LIN {X 0,Y 516.467,Z 235.214,A -85,B 0,C 180,E1 -4935.822,E2 -4935.822} C_VEL
LIN {X 0,Y 516.489,Z 231.626,A -85,B 0,C 180,E1 -4939.019,E2 -4939.019} C_VEL
LIN {X 0,Y 516.548,Z 228.079,A -85,B 0,C 180,E1 -4942.181,E2 -4942.181} C_VEL
LIN {X 0,Y 516.558,Z 225.48,A -85,B 0,C 180,E1 -4944.536,E2 -4944.536} C_VEL
LIN {X 0,Y 516.606,Z 224.598,A -85,B 0,C 180,E1 -4945.319,E2 -4945.319} C_VEL
LIN {X 0,Y 516.602,Z 224.14,A -85,B 0,C 180,E1 -4946.1,E2 -4946.1} C_VEL
LIN {X 0,Y 516.939,Z 224.095,A -85,B 0,C 180,E1 -4948.443,E2 -4948.443} C_VEL
LIN {X 0,Y 517.084,Z 224.078,A -85,B 0,C 180,E1 -4950.78,E2 -4950.78} C_VEL
LIN {X 0,Y 517.003,Z 224.088,A -85,B 0,C 180,E1 -4953.118,E2 -4953.118} C_VEL
LIN {X 0,Y 516.997,Z 224.088,A -85,B 0,C 180,E1 -4956.244,E2 -4956.244} C_VEL
LIN {X 0,Y 516.948,Z 224.094,A -85,B 0,C 180,E1 -4959.39,E2 -4959.39} C_VEL
LIN {X 0,Y 516.969,Z 224.092,A -85,B 0,C 180,E1 -4961.825,E2 -4961.825} C_VEL
LIN {X 0,Y 516.931,Z 224.096,A -85,B 0,C 180,E1 -4965.148,E2 -4965.148} C_VEL
LIN {X 0,Y 516.914,Z 224.097,A -85,B 0,C 180,E1 -4968.223,E2 -4968.223} C_VEL
LIN {X 0,Y 516.903,Z 224.099,A -85,B 0,C 180,E1 -4970.703,E2 -4970.703} C_VEL
LIN {X 0,Y 516.881,Z 224.103,A -85,B 0,C 180,E1 -4973.224,E2 -4973.224} C_VEL
LIN {X 0,Y 516.934,Z 224.095,A -85,B 0,C 180,E1 -4976.198,E2 -4976.198} C_VEL
LIN {X 0,Y 516.912,Z 224.098,A -85,B 0,C 180,E1 -4979.306,E2 -4979.306} C_VEL
LIN {X 0,Y 516.892,Z 224.101,A -85,B 0,C 180,E1 -4982.546,E2 -4982.546} C_VEL
LIN {X 0,Y 516.875,Z 224.102,A -85,B 0,C 180,E1 -4985.334,E2 -4985.334} C_VEL
LIN {X 0,Y 516.874,Z 224.101,A -85,B 0,C 180,E1 -4987.945,E2 -4987.945} C_VEL
LIN {X 0,Y 516.897,Z 224.101,A -85,B 0,C 180,E1 -4990.741,E2 -4990.741} C_VEL
LIN {X 0,Y 516.877,Z 224.102,A -85,B 0,C 180,E1 -4993.905,E2 -4993.905} C_VEL
LIN {X 0,Y 516.877,Z 224.102,A -85,B 0,C 180,E1 -4996.109,E2 -4996.109} C_VEL
LIN {X 0,Y 516.9,Z 224.098,A -85,B 0,C 180,E1 -4999.262,E2 -4999.262} C_VEL
LIN {X 0,Y 516.878,Z 224.103,A -85,B 0,C 180,E1 -5002.058,E2 -5002.058} C_VEL
LIN {X 0,Y 516.89,Z 224.1,A -85,B 0,C 180,E1 -5005.178,E2 -5005.178} C_VEL
LIN {X 0,Y 516.875,Z 224.104,A -85,B 0,C 180,E1 -5007.977,E2 -5007.977} C_VEL
LIN {X 0,Y 516.921,Z 224.096,A -85,B 0,C 180,E1 -5010.697,E2 -5010.697} C_VEL
LIN {X 0,Y 516.943,Z 224.095,A -85,B 0,C 180,E1 -5013.806,E2 -5013.806} C_VEL
LIN {X 0,Y 516.861,Z 224.106,A -85,B 0,C 180,E1 -5016.778,E2 -5016.778} C_VEL
LIN {X 0,Y 516.942,Z 224.094,A -85,B 0,C 180,E1 -5019.733,E2 -5019.733} C_VEL
LIN {X 0,Y 516.922,Z 224.098,A -85,B 0,C 180,E1 -5022.597,E2 -5022.597} C_VEL
LIN {X 0,Y 516.946,Z 224.094,A -85,B 0,C 180,E1 -5025.032,E2 -5025.032} C_VEL
LIN {X 0,Y 517.01,Z 224.087,A -85,B 0,C 180,E1 -5028.236,E2 -5028.236} C_VEL
LIN {X 0,Y 516.96,Z 224.091,A -85,B 0,C 180,E1 -5031.401,E2 -5031.401} C_VEL
LIN {X 0,Y 517.015,Z 224.085,A -85,B 0,C 180,E1 -5033.758,E2 -5033.758} C_VEL
LIN {X 0,Y 517.085,Z 224.078,A -85,B 0,C 180,E1 -5037.664,E2 -5037.664} C_VEL
LIN {X 0,Y 517.098,Z 224.075,A -85,B 0,C 180,E1 -5040.78,E2 -5040.78} C_VEL
LIN {X 0,Y 516.992,Z 224.087,A -85,B 0,C 180,E1 -5043.118,E2 -5043.118} C_VEL
LIN {X 0,Y 517.008,Z 224.086,A -85,B 0,C 180,E1 -5046.244,E2 -5046.244} C_VEL
LIN {X 0,Y 516.949,Z 224.094,A -85,B 0,C 180,E1 -5049.39,E2 -5049.39} C_VEL
LIN {X 0,Y 516.961,Z 224.092,A -85,B 0,C 180,E1 -5051.808,E2 -5051.808} C_VEL
LIN {X 0,Y 516.952,Z 224.093,A -85,B 0,C 180,E1 -5055.146,E2 -5055.146} C_VEL
LIN {X 0,Y 516.921,Z 224.097,A -85,B 0,C 180,E1 -5058.223,E2 -5058.223} C_VEL
LIN {X 0,Y 516.921,Z 224.098,A -85,B 0,C 180,E1 -5060.702,E2 -5060.702} C_VEL
LIN {X 0,Y 516.894,Z 224.1,A -85,B 0,C 180,E1 -5064.074,E2 -5064.074} C_VEL
LIN {X 0,Y 516.915,Z 224.097,A -85,B 0,C 180,E1 -5066.659,E2 -5066.659} C_VEL
LIN {X 0,Y 516.918,Z 224.099,A -85,B 0,C 180,E1 -5069.524,E2 -5069.524} C_VEL
LIN {X 0,Y 516.903,Z 224.098,A -85,B 0,C 180,E1 -5072.543,E2 -5072.543} C_VEL
LIN {X 0,Y 516.874,Z 224.105,A -85,B 0,C 180,E1 -5075.33,E2 -5075.33} C_VEL
LIN {X 0,Y 516.888,Z 224.1,A -85,B 0,C 180,E1 -5077.943,E2 -5077.943} C_VEL
LIN {X 0,Y 516.892,Z 224.1,A -85,B 0,C 180,E1 -5080.742,E2 -5080.742} C_VEL
LIN {X 0,Y 516.891,Z 224.1,A -85,B 0,C 180,E1 -5082.832,E2 -5082.832} C_VEL
LIN {X 0,Y 516.904,Z 224.097,A -85,B 0,C 180,E1 -5085.007,E2 -5085.007} C_VEL
LIN {X 0,Y 516.922,Z 224.096,A -85,B 0,C 180,E1 -5088.399,E2 -5088.399} C_VEL
LIN {X 0,Y 516.91,Z 224.226,A -85,B 0,C 180,E1 -5091.385,E2 -5091.385} C_VEL
LIN {X 0,Y 517.907,Z 230.288,A -85,B 0,C 180,E1 -5093.821,E2 -5093.821} C_VEL
LIN {X 0,Y 517.949,Z 235.762,A -85,B 0,C 180,E1 -5095.865,E2 -5095.865} C_VEL
LIN {X 0,Y 517.702,Z 243.001,A -85,B 0,C 180,E1 -5098.462,E2 -5098.462} C_VEL
LIN {X 0,Y 517.337,Z 252.149,A -85,B 0,C 180,E1 -5101.609,E2 -5101.609} C_VEL
LIN {X 0,Y 517.129,Z 261.34,A -85,B 0,C 180,E1 -5104.652,E2 -5104.652} C_VEL
LIN {X 0,Y 516.921,Z 270.537,A -85,B 0,C 180,E1 -5107.623,E2 -5107.623} C_VEL
LIN {X 0,Y 516.769,Z 279.876,A -85,B 0,C 180,E1 -5110.536,E2 -5110.536} C_VEL
LIN {X 0,Y 516.6,Z 290.693,A -85,B 0,C 180,E1 -5113.805,E2 -5113.805} C_VEL
LIN {X 0,Y 516.522,Z 298.272,A -85,B 0,C 180,E1 -5116.099,E2 -5116.099} C_VEL
LIN {X 0,Y 518.346,Z 310.965,A -85,B 0,C 180,E1 -5116.436,E2 -5116.436} C_VEL
LIN {X 0,Y 518.162,Z 323.395,A -85,B 0,C 180,E1 -5116.868,E2 -5116.868} C_VEL
LIN {X 0,Y 517.868,Z 335.653,A -85,B 0,C 180,E1 -5117.458,E2 -5117.458} C_VEL
LIN {X 0,Y 517.559,Z 346.352,A -85,B 0,C 180,E1 -5118.121,E2 -5118.121} C_VEL
LIN {X 0,Y 517.314,Z 356.898,A -85,B 0,C 180,E1 -5118.936,E2 -5118.936} C_VEL
LIN {X 0,Y 517.031,Z 366.256,A -85,B 0,C 180,E1 -5119.821,E2 -5119.821} C_VEL
LIN {X 0,Y 516.801,Z 374.794,A -85,B 0,C 180,E1 -5120.805,E2 -5120.805} C_VEL
LIN {X 0,Y 516.587,Z 383.122,A -85,B 0,C 180,E1 -5121.983,E2 -5121.983} C_VEL
LIN {X 0,Y 516.441,Z 390.084,A -85,B 0,C 180,E1 -5123.208,E2 -5123.208} C_VEL
LIN {X 0,Y 516.397,Z 395.989,A -85,B 0,C 180,E1 -5124.532,E2 -5124.532} C_VEL
LIN {X 0,Y 516.314,Z 399.982,A -85,B 0,C 180,E1 -5125.706,E2 -5125.706} C_VEL
LIN {X 0,Y 516.283,Z 402.931,A -85,B 0,C 180,E1 -5126.878,E2 -5126.878} C_VEL
LIN {X 0,Y 516.262,Z 404.335,A -85,B 0,C 180,E1 -5127.659,E2 -5127.659} C_VEL
LIN {X 0,Y 516.166,Z 405.942,A -85,B 0,C 180,E1 -5129.219,E2 -5129.219} C_VEL
LIN {X 0,Y 516.166,Z 406.157,A -85,B 0,C 180,E1 -5129.999,E2 -5129.999} C_VEL
LIN {X 0,Y 516.192,Z 405.326,A -85,B 0,C 180,E1 -5131.56,E2 -5131.56} C_VEL
LIN {X 0,Y 516.262,Z 404.325,A -85,B 0,C 180,E1 -5132.34,E2 -5132.34} C_VEL
LIN {X 0,Y 516.283,Z 402.917,A -85,B 0,C 180,E1 -5133.121,E2 -5133.121} C_VEL
LIN {X 0,Y 516.313,Z 399.957,A -85,B 0,C 180,E1 -5134.293,E2 -5134.293} C_VEL
LIN {X 0,Y 516.397,Z 395.952,A -85,B 0,C 180,E1 -5135.466,E2 -5135.466} C_VEL
LIN {X 0,Y 516.473,Z 390.048,A -85,B 0,C 180,E1 -5136.788,E2 -5136.788} C_VEL
LIN {X 0,Y 516.586,Z 383.063,A -85,B 0,C 180,E1 -5138.015,E2 -5138.015} C_VEL
LIN {X 0,Y 516.8,Z 374.717,A -85,B 0,C 180,E1 -5139.194,E2 -5139.194} C_VEL
LIN {X 0,Y 517,Z 366.163,A -85,B 0,C 180,E1 -5140.178,E2 -5140.178} C_VEL
LIN {X 0,Y 517.346,Z 355.609,A -85,B 0,C 180,E1 -5141.161,E2 -5141.161} C_VEL
LIN {X 0,Y 517.589,Z 343.972,A -85,B 0,C 180,E1 -5142.033,E2 -5142.033} C_VEL
LIN {X 0,Y 517.92,Z 331.793,A -85,B 0,C 180,E1 -5142.738,E2 -5142.738} C_VEL
LIN {X 0,Y 518.206,Z 319.398,A -85,B 0,C 180,E1 -5143.279,E2 -5143.279} C_VEL
LIN {X 0,Y 518.231,Z 310.339,A -85,B 0,C 180,E1 -5143.578,E2 -5143.578} C_VEL
LIN {X 0,Y 516.503,Z 297.887,A -85,B 0,C 180,E1 -5143.925,E2 -5143.925} C_VEL
LIN {X 0,Y 516.582,Z 288.976,A -85,B 0,C 180,E1 -5146.6,E2 -5146.6} C_VEL
LIN {X 0,Y 516.745,Z 279.489,A -85,B 0,C 180,E1 -5149.463,E2 -5149.463} C_VEL
LIN {X 0,Y 516.901,Z 269.991,A -85,B 0,C 180,E1 -5152.397,E2 -5152.397} C_VEL
LIN {X 0,Y 517.058,Z 260.81,A -85,B 0,C 180,E1 -5155.35,E2 -5155.35} C_VEL
LIN {X 0,Y 517.258,Z 251.656,A -85,B 0,C 180,E1 -5158.394,E2 -5158.394} C_VEL
LIN {X 0,Y 517.556,Z 243.591,A -85,B 0,C 180,E1 -5161.185,E2 -5161.185} C_VEL
LIN {X 0,Y 517.842,Z 236.392,A -85,B 0,C 180,E1 -5163.809,E2 -5163.809} C_VEL
LIN {X 0,Y 518.004,Z 231.462,A -85,B 0,C 180,E1 -5165.689,E2 -5165.689} C_VEL
LIN {X 0,Y 517.334,Z 226.619,A -85,B 0,C 180,E1 -5167.684,E2 -5167.684} C_VEL
LIN {X 0,Y 516.882,Z 224.103,A -85,B 0,C 180,E1 -5168.834,E2 -5168.834} C_VEL
LIN {X 0,Y 516.915,Z 224.098,A -85,B 0,C 180,E1 -5171.774,E2 -5171.774} C_VEL
LIN {X 0,Y 516.894,Z 224.101,A -85,B 0,C 180,E1 -5175.006,E2 -5175.006} C_VEL
LIN {X 0,Y 516.916,Z 224.098,A -85,B 0,C 180,E1 -5178.397,E2 -5178.397} C_VEL
LIN {X 0,Y 516.88,Z 224.103,A -85,B 0,C 180,E1 -5181.283,E2 -5181.283} C_VEL
LIN {X 0,Y 516.886,Z 224.102,A -85,B 0,C 180,E1 -5184.22,E2 -5184.22} C_VEL
LIN {X 0,Y 516.894,Z 224.101,A -85,B 0,C 180,E1 -5187.052,E2 -5187.052} C_VEL
LIN {X 0,Y 516.889,Z 224.101,A -85,B 0,C 180,E1 -5189.795,E2 -5189.795} C_VEL
LIN {X 0,Y 516.927,Z 224.098,A -85,B 0,C 180,E1 -5192.466,E2 -5192.466} C_VEL
LIN {X 0,Y 516.872,Z 224.103,A -85,B 0,C 180,E1 -5195.069,E2 -5195.069} C_VEL
LIN {X 0,Y 516.865,Z 224.103,A -85,B 0,C 180,E1 -5197.62,E2 -5197.62} C_VEL
LIN {X 0,Y 516.929,Z 224.096,A -85,B 0,C 180,E1 -5200.129,E2 -5200.129} C_VEL
LIN {X 0,Y 516.926,Z 224.098,A -85,B 0,C 180,E1 -5202.595,E2 -5202.595} C_VEL
LIN {X 0,Y 516.938,Z 224.096,A -85,B 0,C 180,E1 -5205.029,E2 -5205.029} C_VEL
LIN {X 0,Y 517,Z 224.089,A -85,B 0,C 180,E1 -5208.233,E2 -5208.233} C_VEL
LIN {X 0,Y 516.965,Z 224.092,A -85,B 0,C 180,E1 -5211.399,E2 -5211.399} C_VEL
LIN {X 0,Y 517.007,Z 224.087,A -85,B 0,C 180,E1 -5213.756,E2 -5213.756} C_VEL
LIN {X 0,Y 517.077,Z 224.078,A -85,B 0,C 180,E1 -5217.662,E2 -5217.662} C_VEL
LIN {X 0,Y 517.09,Z 224.078,A -85,B 0,C 180,E1 -5220.778,E2 -5220.778} C_VEL
LIN {X 0,Y 517.01,Z 224.087,A -85,B 0,C 180,E1 -5223.116,E2 -5223.116} C_VEL
LIN {X 0,Y 517.004,Z 224.088,A -85,B 0,C 180,E1 -5226.242,E2 -5226.242} C_VEL
LIN {X 0,Y 516.953,Z 224.093,A -85,B 0,C 180,E1 -5229.388,E2 -5229.388} C_VEL
LIN {X 0,Y 516.975,Z 224.091,A -85,B 0,C 180,E1 -5231.823,E2 -5231.823} C_VEL
LIN {X 0,Y 516.935,Z 224.097,A -85,B 0,C 180,E1 -5235.145,E2 -5235.145} C_VEL
LIN {X 0,Y 516.859,Z 224.108,A -85,B 0,C 180,E1 -5237.86,E2 -5237.86} C_VEL
LIN {X 0,Y 516.643,Z 224.391,A -85,B 0,C 180,E1 -5239.88,E2 -5239.88} C_VEL
LIN {X 0,Y 516.601,Z 227.102,A -85,B 0,C 180,E1 -5242.389,E2 -5242.389} C_VEL
LIN {X 0,Y 516.556,Z 229.906,A -85,B 0,C 180,E1 -5244.945,E2 -5244.945} C_VEL
LIN {X 0,Y 516.491,Z 233.036,A -85,B 0,C 180,E1 -5247.816,E2 -5247.816} C_VEL
LIN {X 0,Y 516.431,Z 236.511,A -85,B 0,C 180,E1 -5250.981,E2 -5250.981} C_VEL
LIN {X 0,Y 516.357,Z 239.775,A -85,B 0,C 180,E1 -5253.918,E2 -5253.918} C_VEL
LIN {X 0,Y 516.278,Z 242.962,A -85,B 0,C 180,E1 -5256.794,E2 -5256.794} C_VEL
LIN {X 0,Y 516.297,Z 245.663,A -85,B 0,C 180,E1 -5259.199,E2 -5259.199} C_VEL
LIN {X 0,Y 518.486,Z 256.449,A -85,B 0,C 180,E1 -5259.549,E2 -5259.549} C_VEL
LIN {X 0,Y 518.293,Z 269.265,A -85,B 0,C 180,E1 -5260.032,E2 -5260.032} C_VEL
LIN {X 0,Y 517.996,Z 281.061,A -85,B 0,C 180,E1 -5260.633,E2 -5260.633} C_VEL
LIN {X 0,Y 517.716,Z 291.239,A -85,B 0,C 180,E1 -5261.298,E2 -5261.298} C_VEL
LIN {X 0,Y 517.48,Z 301.242,A -85,B 0,C 180,E1 -5262.109,E2 -5262.109} C_VEL
LIN {X 0,Y 517.178,Z 310.969,A -85,B 0,C 180,E1 -5263.08,E2 -5263.08} C_VEL
LIN {X 0,Y 516.902,Z 319.892,A -85,B 0,C 180,E1 -5264.177,E2 -5264.177} C_VEL
LIN {X 0,Y 516.877,Z 320.67,A -85,B 0,C 180,E1 -5264.286,E2 -5264.286} C_VEL
LIN {X 0,Y 516.11,Z 324.315,A -85,B 0,C 180,E1 -5264.8,E2 -5264.8} C_VEL
LIN {X 0,Y 511.766,Z 331.837,A -85,B 0,C 180,E1 -5266.008,E2 -5266.008} C_VEL
LIN {X 0,Y 509.733,Z 335.586,A -85,B 0,C 180,E1 -5266.757,E2 -5266.757} C_VEL
LIN {X 0,Y 509.375,Z 337.272,A -85,B 0,C 180,E1 -5267.155,E2 -5267.155} C_VEL
LIN {X 0,Y 509.29,Z 342.03,A -85,B 0,C 180,E1 -5268.519,E2 -5268.519} C_VEL
LIN {X 0,Y 509.243,Z 344.721,A -85,B 0,C 180,E1 -5269.562,E2 -5269.562} C_VEL
LIN {X 0,Y 509.148,Z 346.72,A -85,B 0,C 180,E1 -5270.621,E2 -5270.621} C_VEL
LIN {X 0,Y 509.089,Z 348.144,A -85,B 0,C 180,E1 -5271.893,E2 -5271.893} C_VEL
LIN {X 0,Y 509.085,Z 348.541,A -85,B 0,C 180,E1 -5273.194,E2 -5273.194} C_VEL
LIN {X 0,Y 509.077,Z 347.811,A -85,B 0,C 180,E1 -5274.563,E2 -5274.563} C_VEL
LIN {X 0,Y 509.164,Z 345.936,A -85,B 0,C 180,E1 -5275.909,E2 -5275.909} C_VEL
LIN {X 0,Y 509.23,Z 342.382,A -85,B 0,C 180,E1 -5277.437,E2 -5277.437} C_VEL
LIN {X 0,Y 509.359,Z 337.714,A -85,B 0,C 180,E1 -5278.807,E2 -5278.807} C_VEL
LIN {X 0,Y 509.544,Z 331.262,A -85,B 0,C 180,E1 -5280.23,E2 -5280.23} C_VEL
LIN {X 0,Y 509.748,Z 324.793,A -85,B 0,C 180,E1 -5281.355,E2 -5281.355} C_VEL
LIN {X 0,Y 509.989,Z 316.614,A -85,B 0,C 180,E1 -5282.507,E2 -5282.507} C_VEL
LIN {X 0,Y 510.276,Z 307.618,A -85,B 0,C 180,E1 -5283.535,E2 -5283.535} C_VEL
LIN {X 0,Y 510.638,Z 296.904,A -85,B 0,C 180,E1 -5284.527,E2 -5284.527} C_VEL
LIN {X 0,Y 510.951,Z 285.423,A -85,B 0,C 180,E1 -5285.367,E2 -5285.367} C_VEL
LIN {X 0,Y 511.25,Z 272.908,A -85,B 0,C 180,E1 -5286.077,E2 -5286.077} C_VEL
LIN {X 0,Y 511.593,Z 260.24,A -85,B 0,C 180,E1 -5286.604,E2 -5286.604} C_VEL
LIN {X 0,Y 511.386,Z 255.913,A -85,B 0,C 180,E1 -5286.755,E2 -5286.755} C_VEL
LIN {X 0,Y 509.252,Z 245.771,A -85,B 0,C 180,E1 -5287.081,E2 -5287.081} C_VEL
LIN {X 0,Y 509.288,Z 242.619,A -85,B 0,C 180,E1 -5289.82,E2 -5289.82} C_VEL
LIN {X 0,Y 509.338,Z 239.772,A -85,B 0,C 180,E1 -5292.329,E2 -5292.329} C_VEL
LIN {X 0,Y 509.409,Z 236.06,A -85,B 0,C 180,E1 -5295.622,E2 -5295.622} C_VEL
LIN {X 0,Y 509.422,Z 232.451,A -85,B 0,C 180,E1 -5298.864,E2 -5298.864} C_VEL
LIN {X 0,Y 509.487,Z 228.868,A -85,B 0,C 180,E1 -5302.072,E2 -5302.072} C_VEL
LIN {X 0,Y 509.488,Z 226.23,A -85,B 0,C 180,E1 -5304.46,E2 -5304.46} C_VEL
LIN {X 0,Y 509.545,Z 225.354,A -85,B 0,C 180,E1 -5305.254,E2 -5305.254} C_VEL
LIN {X 0,Y 509.597,Z 225.012,A -85,B 0,C 180,E1 -5306.838,E2 -5306.838} C_VEL
LIN {X 0,Y 509.904,Z 224.971,A -85,B 0,C 180,E1 -5308.421,E2 -5308.421} C_VEL
LIN {X 0,Y 510.053,Z 224.954,A -85,B 0,C 180,E1 -5310.79,E2 -5310.79} C_VEL
LIN {X 0,Y 509.945,Z 224.967,A -85,B 0,C 180,E1 -5313.161,E2 -5313.161} C_VEL
LIN {X 0,Y 509.965,Z 224.963,A -85,B 0,C 180,E1 -5316.331,E2 -5316.331} C_VEL
LIN {X 0,Y 509.907,Z 224.972,A -85,B 0,C 180,E1 -5318.721,E2 -5318.721} C_VEL
LIN {X 0,Y 509.937,Z 224.967,A -85,B 0,C 180,E1 -5321.932,E2 -5321.932} C_VEL
LIN {X 0,Y 509.88,Z 224.975,A -85,B 0,C 180,E1 -5325.243,E2 -5325.243} C_VEL
LIN {X 0,Y 509.876,Z 224.974,A -85,B 0,C 180,E1 -5328.002,E2 -5328.002} C_VEL
LIN {X 0,Y 509.846,Z 224.979,A -85,B 0,C 180,E1 -5331.003,E2 -5331.003} C_VEL
LIN {X 0,Y 509.839,Z 224.979,A -85,B 0,C 180,E1 -5333.564,E2 -5333.564} C_VEL
LIN {X 0,Y 509.903,Z 224.97,A -85,B 0,C 180,E1 -5336.381,E2 -5336.381} C_VEL
LIN {X 0,Y 509.867,Z 224.976,A -85,B 0,C 180,E1 -5338.846,E2 -5338.846} C_VEL
LIN {X 0,Y 509.816,Z 224.982,A -85,B 0,C 180,E1 -5341.591,E2 -5341.591} C_VEL
LIN {X 0,Y 509.846,Z 224.978,A -85,B 0,C 180,E1 -5344.415,E2 -5344.415} C_VEL
LIN {X 0,Y 509.811,Z 224.982,A -85,B 0,C 180,E1 -5347.342,E2 -5347.342} C_VEL
LIN {X 0,Y 509.854,Z 224.977,A -85,B 0,C 180,E1 -5350.382,E2 -5350.382} C_VEL
LIN {X 0,Y 509.834,Z 224.98,A -85,B 0,C 180,E1 -5353.066,E2 -5353.066} C_VEL
LIN {X 0,Y 509.825,Z 224.98,A -85,B 0,C 180,E1 -5355.794,E2 -5355.794} C_VEL
LIN {X 0,Y 509.861,Z 224.978,A -85,B 0,C 180,E1 -5358.577,E2 -5358.577} C_VEL
LIN {X 0,Y 509.855,Z 224.975,A -85,B 0,C 180,E1 -5361.665,E2 -5361.665} C_VEL
LIN {X 0,Y 509.841,Z 224.979,A -85,B 0,C 180,E1 -5364.625,E2 -5364.625} C_VEL
LIN {X 0,Y 509.861,Z 224.975,A -85,B 0,C 180,E1 -5367.483,E2 -5367.483} C_VEL
LIN {X 0,Y 509.857,Z 224.978,A -85,B 0,C 180,E1 -5370.275,E2 -5370.275} C_VEL
LIN {X 0,Y 509.885,Z 224.972,A -85,B 0,C 180,E1 -5372.946,E2 -5372.946} C_VEL
LIN {X 0,Y 509.852,Z 224.976,A -85,B 0,C 180,E1 -5375.575,E2 -5375.575} C_VEL
LIN {X 0,Y 509.824,Z 224.983,A -85,B 0,C 180,E1 -5378.15,E2 -5378.15} C_VEL
LIN {X 0,Y 509.866,Z 224.975,A -85,B 0,C 180,E1 -5380.683,E2 -5380.683} C_VEL
LIN {X 0,Y 509.882,Z 224.972,A -85,B 0,C 180,E1 -5383.176,E2 -5383.176} C_VEL
LIN {X 0,Y 509.868,Z 224.975,A -85,B 0,C 180,E1 -5385.636,E2 -5385.636} C_VEL
LIN {X 0,Y 509.926,Z 224.966,A -85,B 0,C 180,E1 -5388.876,E2 -5388.876} C_VEL
LIN {X 0,Y 509.926,Z 224.969,A -85,B 0,C 180,E1 -5392.079,E2 -5392.079} C_VEL
LIN {X 0,Y 509.986,Z 224.96,A -85,B 0,C 180,E1 -5394.466,E2 -5394.466} C_VEL
LIN {X 0,Y 510.057,Z 224.954,A -85,B 0,C 180,E1 -5397.632,E2 -5397.632} C_VEL
LIN {X 0,Y 510.062,Z 224.952,A -85,B 0,C 180,E1 -5400.001,E2 -5400.001} C_VEL
LIN {X 0,Y 510.057,Z 224.951,A -85,B 0,C 180,E1 -5402.37,E2 -5402.37} C_VEL
LIN {X 0,Y 509.959,Z 224.964,A -85,B 0,C 180,E1 -5406.331,E2 -5406.331} C_VEL
LIN {X 0,Y 509.912,Z 224.969,A -85,B 0,C 180,E1 -5408.721,E2 -5408.721} C_VEL
LIN {X 0,Y 509.913,Z 224.97,A -85,B 0,C 180,E1 -5411.933,E2 -5411.933} C_VEL
LIN {X 0,Y 509.903,Z 224.971,A -85,B 0,C 180,E1 -5415.243,E2 -5415.243} C_VEL
LIN {X 0,Y 509.866,Z 224.975,A -85,B 0,C 180,E1 -5418.485,E2 -5418.485} C_VEL
LIN {X 0,Y 509.859,Z 224.976,A -85,B 0,C 180,E1 -5421.002,E2 -5421.002} C_VEL
LIN {X 0,Y 509.828,Z 224.981,A -85,B 0,C 180,E1 -5423.565,E2 -5423.565} C_VEL
LIN {X 0,Y 509.883,Z 224.974,A -85,B 0,C 180,E1 -5427.057,E2 -5427.057} C_VEL
LIN {X 0,Y 509.866,Z 224.975,A -85,B 0,C 180,E1 -5429.751,E2 -5429.751} C_VEL
LIN {X 0,Y 509.876,Z 224.974,A -85,B 0,C 180,E1 -5432.773,E2 -5432.773} C_VEL
LIN {X 0,Y 509.834,Z 224.979,A -85,B 0,C 180,E1 -5435.578,E2 -5435.578} C_VEL
LIN {X 0,Y 509.857,Z 224.975,A -85,B 0,C 180,E1 -5438.338,E2 -5438.338} C_VEL
LIN {X 0,Y 509.864,Z 224.975,A -85,B 0,C 180,E1 -5441.426,E2 -5441.426} C_VEL
LIN {X 0,Y 509.848,Z 224.978,A -85,B 0,C 180,E1 -5444.67,E2 -5444.67} C_VEL
LIN {X 0,Y 509.864,Z 224.975,A -85,B 0,C 180,E1 -5448.103,E2 -5448.103} C_VEL
LIN {X 0,Y 509.879,Z 225.144,A -85,B 0,C 180,E1 -5451.158,E2 -5451.158} C_VEL
LIN {X 0,Y 510.933,Z 231.463,A -85,B 0,C 180,E1 -5453.737,E2 -5453.737} C_VEL
LIN {X 0,Y 510.988,Z 236.566,A -85,B 0,C 180,E1 -5455.673,E2 -5455.673} C_VEL
LIN {X 0,Y 510.686,Z 244.227,A -85,B 0,C 180,E1 -5458.469,E2 -5458.469} C_VEL
LIN {X 0,Y 510.378,Z 251.989,A -85,B 0,C 180,E1 -5461.186,E2 -5461.186} C_VEL
LIN {X 0,Y 510.125,Z 261.115,A -85,B 0,C 180,E1 -5464.279,E2 -5464.279} C_VEL
LIN {X 0,Y 509.881,Z 270.771,A -85,B 0,C 180,E1 -5467.445,E2 -5467.445} C_VEL
LIN {X 0,Y 509.715,Z 279.602,A -85,B 0,C 180,E1 -5470.256,E2 -5470.256} C_VEL
LIN {X 0,Y 509.533,Z 290.304,A -85,B 0,C 180,E1 -5473.574,E2 -5473.574} C_VEL
LIN {X 0,Y 509.424,Z 297.841,A -85,B 0,C 180,E1 -5475.901,E2 -5475.901} C_VEL
LIN {X 0,Y 511.3,Z 310.989,A -85,B 0,C 180,E1 -5476.258,E2 -5476.258} C_VEL
LIN {X 0,Y 511.352,Z 319.154,A -85,B 0,C 180,E1 -5476.538,E2 -5476.538} C_VEL
LIN {X 0,Y 510.987,Z 331.525,A -85,B 0,C 180,E1 -5477.085,E2 -5477.085} C_VEL
LIN {X 0,Y 510.695,Z 342.32,A -85,B 0,C 180,E1 -5477.71,E2 -5477.71} C_VEL
LIN {X 0,Y 510.412,Z 352.944,A -85,B 0,C 180,E1 -5478.482,E2 -5478.482} C_VEL
LIN {X 0,Y 510.069,Z 363.893,A -85,B 0,C 180,E1 -5479.48,E2 -5479.48} C_VEL
LIN {X 0,Y 509.789,Z 372.791,A -85,B 0,C 180,E1 -5480.477,E2 -5480.477} C_VEL
LIN {X 0,Y 509.575,Z 381.48,A -85,B 0,C 180,E1 -5481.673,E2 -5481.673} C_VEL
LIN {X 0,Y 509.41,Z 388.422,A -85,B 0,C 180,E1 -5482.867,E2 -5482.867} C_VEL
LIN {X 0,Y 509.314,Z 393.988,A -85,B 0,C 180,E1 -5484.059,E2 -5484.059} C_VEL
LIN {X 0,Y 509.187,Z 398.35,A -85,B 0,C 180,E1 -5485.249,E2 -5485.249} C_VEL
LIN {X 0,Y 509.276,Z 400.666,A -85,B 0,C 180,E1 -5486.043,E2 -5486.043} C_VEL
LIN {X 0,Y 509.202,Z 402.535,A -85,B 0,C 180,E1 -5486.834,E2 -5486.834} C_VEL
LIN {X 0,Y 509.191,Z 403.94,A -85,B 0,C 180,E1 -5487.626,E2 -5487.626} C_VEL
LIN {X 0,Y 509.079,Z 405.544,A -85,B 0,C 180,E1 -5489.208,E2 -5489.208} C_VEL
LIN {X 0,Y 509.078,Z 405.759,A -85,B 0,C 180,E1 -5489.999,E2 -5489.999} C_VEL
LIN {X 0,Y 509.113,Z 404.926,A -85,B 0,C 180,E1 -5491.581,E2 -5491.581} C_VEL
LIN {X 0,Y 509.19,Z 403.923,A -85,B 0,C 180,E1 -5492.372,E2 -5492.372} C_VEL
LIN {X 0,Y 509.202,Z 402.511,A -85,B 0,C 180,E1 -5493.164,E2 -5493.164} C_VEL
LIN {X 0,Y 509.207,Z 399.546,A -85,B 0,C 180,E1 -5494.353,E2 -5494.353} C_VEL
LIN {X 0,Y 509.309,Z 395.538,A -85,B 0,C 180,E1 -5495.542,E2 -5495.542} C_VEL
LIN {X 0,Y 509.408,Z 389.475,A -85,B 0,C 180,E1 -5496.913,E2 -5496.913} C_VEL
LIN {X 0,Y 509.509,Z 382.635,A -85,B 0,C 180,E1 -5498.127,E2 -5498.127} C_VEL
LIN {X 0,Y 509.744,Z 374.284,A -85,B 0,C 180,E1 -5499.322,E2 -5499.322} C_VEL
LIN {X 0,Y 509.972,Z 365.724,A -85,B 0,C 180,E1 -5500.32,E2 -5500.32} C_VEL
LIN {X 0,Y 510.356,Z 355.163,A -85,B 0,C 180,E1 -5501.316,E2 -5501.316} C_VEL
LIN {X 0,Y 510.599,Z 343.519,A -85,B 0,C 180,E1 -5502.2,E2 -5502.2} C_VEL
LIN {X 0,Y 510.988,Z 331.333,A -85,B 0,C 180,E1 -5502.914,E2 -5502.914} C_VEL
LIN {X 0,Y 511.305,Z 318.936,A -85,B 0,C 180,E1 -5503.462,E2 -5503.462} C_VEL
LIN {X 0,Y 511.27,Z 310.779,A -85,B 0,C 180,E1 -5503.741,E2 -5503.741} C_VEL
LIN {X 0,Y 509.507,Z 298.545,A -85,B 0,C 180,E1 -5504.079,E2 -5504.079} C_VEL
LIN {X 0,Y 509.42,Z 297.45,A -85,B 0,C 180,E1 -5504.123,E2 -5504.123} C_VEL
LIN {X 0,Y 509.513,Z 288.533,A -85,B 0,C 180,E1 -5506.837,E2 -5506.837} C_VEL
LIN {X 0,Y 509.671,Z 279.113,A -85,B 0,C 180,E1 -5509.744,E2 -5509.744} C_VEL
LIN {X 0,Y 509.852,Z 269.739,A -85,B 0,C 180,E1 -5512.703,E2 -5512.703} C_VEL
LIN {X 0,Y 510.03,Z 260.498,A -85,B 0,C 180,E1 -5515.724,E2 -5515.724} C_VEL
LIN {X 0,Y 510.288,Z 251.466,A -85,B 0,C 180,E1 -5518.818,E2 -5518.818} C_VEL
LIN {X 0,Y 510.609,Z 243.801,A -85,B 0,C 180,E1 -5521.535,E2 -5521.535} C_VEL
LIN {X 0,Y 510.923,Z 236.159,A -85,B 0,C 180,E1 -5524.377,E2 -5524.377} C_VEL
LIN {X 0,Y 510.932,Z 231.414,A -85,B 0,C 180,E1 -5526.261,E2 -5526.261} C_VEL
LIN {X 0,Y 509.865,Z 224.978,A -85,B 0,C 180,E1 -5529.063,E2 -5529.063} C_VEL
LIN {X 0,Y 509.859,Z 224.978,A -85,B 0,C 180,E1 -5531.896,E2 -5531.896} C_VEL
LIN {X 0,Y 509.838,Z 224.98,A -85,B 0,C 180,E1 -5535.329,E2 -5535.329} C_VEL
LIN {X 0,Y 509.858,Z 224.978,A -85,B 0,C 180,E1 -5538.574,E2 -5538.574} C_VEL
LIN {X 0,Y 509.85,Z 224.978,A -85,B 0,C 180,E1 -5541.785,E2 -5541.785} C_VEL
LIN {X 0,Y 509.842,Z 224.98,A -85,B 0,C 180,E1 -5544.622,E2 -5544.622} C_VEL
LIN {X 0,Y 509.861,Z 224.976,A -85,B 0,C 180,E1 -5547.48,E2 -5547.48} C_VEL
LIN {X 0,Y 509.856,Z 224.978,A -85,B 0,C 180,E1 -5550.273,E2 -5550.273} C_VEL
LIN {X 0,Y 509.883,Z 224.973,A -85,B 0,C 180,E1 -5552.943,E2 -5552.943} C_VEL
LIN {X 0,Y 509.848,Z 224.979,A -85,B 0,C 180,E1 -5555.572,E2 -5555.572} C_VEL
LIN {X 0,Y 509.819,Z 224.983,A -85,B 0,C 180,E1 -5558.147,E2 -5558.147} C_VEL
LIN {X 0,Y 509.861,Z 224.976,A -85,B 0,C 180,E1 -5560.68,E2 -5560.68} C_VEL
LIN {X 0,Y 509.881,Z 224.973,A -85,B 0,C 180,E1 -5563.174,E2 -5563.174} C_VEL
LIN {X 0,Y 509.861,Z 224.976,A -85,B 0,C 180,E1 -5565.633,E2 -5565.633} C_VEL
LIN {X 0,Y 509.918,Z 224.968,A -85,B 0,C 180,E1 -5568.874,E2 -5568.874} C_VEL
LIN {X 0,Y 509.947,Z 224.965,A -85,B 0,C 180,E1 -5572.077,E2 -5572.077} C_VEL
LIN {X 0,Y 509.979,Z 224.961,A -85,B 0,C 180,E1 -5574.463,E2 -5574.463} C_VEL
LIN {X 0,Y 510.049,Z 224.953,A -85,B 0,C 180,E1 -5577.63,E2 -5577.63} C_VEL
LIN {X 0,Y 510.06,Z 224.953,A -85,B 0,C 180,E1 -5580.788,E2 -5580.788} C_VEL
LIN {X 0,Y 509.952,Z 224.966,A -85,B 0,C 180,E1 -5583.159,E2 -5583.159} C_VEL
LIN {X 0,Y 509.972,Z 224.965,A -85,B 0,C 180,E1 -5586.328,E2 -5586.328} C_VEL
LIN {X 0,Y 509.912,Z 224.971,A -85,B 0,C 180,E1 -5588.719,E2 -5588.719} C_VEL
LIN {X 0,Y 509.943,Z 224.967,A -85,B 0,C 180,E1 -5591.929,E2 -5591.929} C_VEL
LIN {X 0,Y 509.884,Z 224.976,A -85,B 0,C 180,E1 -5595.241,E2 -5595.241} C_VEL
LIN {X 0,Y 509.79,Z 224.988,A -85,B 0,C 180,E1 -5597.969,E2 -5597.969} C_VEL
LIN {X 0,Y 509.618,Z 225.01,A -85,B 0,C 180,E1 -5599.327,E2 -5599.327} C_VEL
LIN {X 0,Y 509.567,Z 225.636,A -85,B 0,C 180,E1 -5600.307,E2 -5600.307} C_VEL
LIN {X 0,Y 509.52,Z 229.172,A -85,B 0,C 180,E1 -5603.577,E2 -5603.577} C_VEL
LIN {X 0,Y 509.441,Z 232.062,A -85,B 0,C 180,E1 -5606.273,E2 -5606.273} C_VEL
LIN {X 0,Y 509.392,Z 234.863,A -85,B 0,C 180,E1 -5608.872,E2 -5608.872} C_VEL
LIN {X 0,Y 509.336,Z 237.916,A -85,B 0,C 180,E1 -5611.622,E2 -5611.622} C_VEL
LIN {X 0,Y 509.261,Z 241.014,A -85,B 0,C 180,E1 -5614.457,E2 -5614.457} C_VEL
LIN {X 0,Y 509.198,Z 244.313,A -85,B 0,C 180,E1 -5617.392,E2 -5617.392} C_VEL
LIN {X 0,Y 509.204,Z 246.111,A -85,B 0,C 180,E1 -5619.011,E2 -5619.011} C_VEL
LIN {X 0,Y 511.562,Z 257.166,A -85,B 0,C 180,E1 -5619.375,E2 -5619.375} C_VEL
LIN {X 0,Y 511.38,Z 270.454,A -85,B 0,C 180,E1 -5619.89,E2 -5619.89} C_VEL
LIN {X 0,Y 511.072,Z 282.72,A -85,B 0,C 180,E1 -5620.54,E2 -5620.54} C_VEL
LIN {X 0,Y 510.699,Z 294.274,A -85,B 0,C 180,E1 -5621.34,E2 -5621.34} C_VEL
LIN {X 0,Y 510.391,Z 305.142,A -85,B 0,C 180,E1 -5622.287,E2 -5622.287} C_VEL
LIN {X 0,Y 510.077,Z 314.944,A -85,B 0,C 180,E1 -5623.36,E2 -5623.36} C_VEL
LIN {X 0,Y 509.804,Z 323.211,A -85,B 0,C 180,E1 -5624.477,E2 -5624.477} C_VEL
LIN {X 0,Y 509.555,Z 331.168,A -85,B 0,C 180,E1 -5625.822,E2 -5625.822} C_VEL
LIN {X 0,Y 509.375,Z 337.272,A -85,B 0,C 180,E1 -5627.155,E2 -5627.155} C_VEL
LIN {X 0,Y 508.655,Z 339.636,A -85,B 0,C 180,E1 -5627.761,E2 -5627.761} C_VEL
LIN {X 0,Y 505.722,Z 343.049,A -85,B 0,C 180,E1 -5628.76,E2 -5628.76} C_VEL
LIN {X 0,Y 503.251,Z 345.255,A -85,B 0,C 180,E1 -5629.583,E2 -5629.583} C_VEL
LIN {X 0,Y 502.166,Z 346.546,A -85,B 0,C 180,E1 -5630.231,E2 -5630.231} C_VEL
LIN {X 0,Y 502.065,Z 346.895,A -85,B 0,C 180,E1 -5630.453,E2 -5630.453} C_VEL
LIN {X 0,Y 502,Z 348.602,A -85,B 0,C 180,E1 -5631.976,E2 -5631.976} C_VEL
LIN {X 0,Y 501.992,Z 348.958,A -85,B 0,C 180,E1 -5632.987,E2 -5632.987} C_VEL
LIN {X 0,Y 501.988,Z 348.478,A -85,B 0,C 180,E1 -5634.29,E2 -5634.29} C_VEL
LIN {X 0,Y 502.072,Z 346.82,A -85,B 0,C 180,E1 -5635.675,E2 -5635.675} C_VEL
LIN {X 0,Y 502.154,Z 343.798,A -85,B 0,C 180,E1 -5637.109,E2 -5637.109} C_VEL
LIN {X 0,Y 502.274,Z 339.206,A -85,B 0,C 180,E1 -5638.595,E2 -5638.595} C_VEL
LIN {X 0,Y 502.414,Z 334.396,A -85,B 0,C 180,E1 -5639.764,E2 -5639.764} C_VEL
LIN {X 0,Y 502.594,Z 328.426,A -85,B 0,C 180,E1 -5640.928,E2 -5640.928} C_VEL
LIN {X 0,Y 502.876,Z 321.098,A -85,B 0,C 180,E1 -5642.085,E2 -5642.085} C_VEL
LIN {X 0,Y 503.154,Z 312.195,A -85,B 0,C 180,E1 -5643.22,E2 -5643.22} C_VEL
LIN {X 0,Y 503.536,Z 302.193,A -85,B 0,C 180,E1 -5644.253,E2 -5644.253} C_VEL
LIN {X 0,Y 503.842,Z 291.403,A -85,B 0,C 180,E1 -5645.148,E2 -5645.148} C_VEL
LIN {X 0,Y 504.229,Z 279.184,A -85,B 0,C 180,E1 -5645.941,E2 -5645.941} C_VEL
LIN {X 0,Y 504.544,Z 266.733,A -85,B 0,C 180,E1 -5646.557,E2 -5646.557} C_VEL
LIN {X 0,Y 504.563,Z 257.315,A -85,B 0,C 180,E1 -5646.908,E2 -5646.908} C_VEL
LIN {X 0,Y 502.173,Z 246.113,A -85,B 0,C 180,E1 -5647.297,E2 -5647.297} C_VEL
LIN {X 0,Y 502.213,Z 242.6,A -85,B 0,C 180,E1 -5650.376,E2 -5650.376} C_VEL
LIN {X 0,Y 502.252,Z 239.729,A -85,B 0,C 180,E1 -5652.912,E2 -5652.912} C_VEL
LIN {X 0,Y 502.318,Z 236.921,A -85,B 0,C 180,E1 -5655.414,E2 -5655.414} C_VEL
LIN {X 0,Y 502.362,Z 233.257,A -85,B 0,C 180,E1 -5658.706,E2 -5658.706} C_VEL
LIN {X 0,Y 502.418,Z 229.663,A -85,B 0,C 180,E1 -5661.96,E2 -5661.96} C_VEL
LIN {X 0,Y 502.503,Z 227.87,A -85,B 0,C 180,E1 -5663.577,E2 -5663.577} C_VEL
LIN {X 0,Y 502.486,Z 226.126,A -85,B 0,C 180,E1 -5665.187,E2 -5665.187} C_VEL
LIN {X 0,Y 502.869,Z 225.847,A -85,B 0,C 180,E1 -5668.399,E2 -5668.399} C_VEL
LIN {X 0,Y 503.023,Z 225.829,A -85,B 0,C 180,E1 -5670.801,E2 -5670.801} C_VEL
LIN {X 0,Y 502.889,Z 225.845,A -85,B 0,C 180,E1 -5673.205,E2 -5673.205} C_VEL
LIN {X 0,Y 502.915,Z 225.842,A -85,B 0,C 180,E1 -5676.42,E2 -5676.42} C_VEL
LIN {X 0,Y 502.865,Z 225.849,A -85,B 0,C 180,E1 -5678.844,E2 -5678.844} C_VEL
LIN {X 0,Y 502.88,Z 225.846,A -85,B 0,C 180,E1 -5682.102,E2 -5682.102} C_VEL
LIN {X 0,Y 502.835,Z 225.853,A -85,B 0,C 180,E1 -5685.401,E2 -5685.401} C_VEL
LIN {X 0,Y 502.834,Z 225.851,A -85,B 0,C 180,E1 -5688.124,E2 -5688.124} C_VEL
LIN {X 0,Y 502.785,Z 225.858,A -85,B 0,C 180,E1 -5691.312,E2 -5691.312} C_VEL
LIN {X 0,Y 502.791,Z 225.855,A -85,B 0,C 180,E1 -5693.915,E2 -5693.915} C_VEL
LIN {X 0,Y 502.87,Z 225.847,A -85,B 0,C 180,E1 -5696.567,E2 -5696.567} C_VEL
LIN {X 0,Y 502.814,Z 225.854,A -85,B 0,C 180,E1 -5699.289,E2 -5699.289} C_VEL
LIN {X 0,Y 502.779,Z 225.857,A -85,B 0,C 180,E1 -5702.086,E2 -5702.086} C_VEL
LIN {X 0,Y 502.802,Z 225.857,A -85,B 0,C 180,E1 -5704.966,E2 -5704.966} C_VEL
LIN {X 0,Y 502.787,Z 225.856,A -85,B 0,C 180,E1 -5707.955,E2 -5707.955} C_VEL
LIN {X 0,Y 502.82,Z 225.853,A -85,B 0,C 180,E1 -5711.067,E2 -5711.067} C_VEL
LIN {X 0,Y 502.776,Z 225.857,A -85,B 0,C 180,E1 -5713.377,E2 -5713.377} C_VEL
LIN {X 0,Y 502.784,Z 225.857,A -85,B 0,C 180,E1 -5715.663,E2 -5715.663} C_VEL
LIN {X 0,Y 502.822,Z 225.852,A -85,B 0,C 180,E1 -5719.006,E2 -5719.006} C_VEL
LIN {X 0,Y 502.794,Z 225.857,A -85,B 0,C 180,E1 -5722.048,E2 -5722.048} C_VEL
LIN {X 0,Y 502.806,Z 225.854,A -85,B 0,C 180,E1 -5725.037,E2 -5725.037} C_VEL
LIN {X 0,Y 502.783,Z 225.859,A -85,B 0,C 180,E1 -5727.917,E2 -5727.917} C_VEL
LIN {X 0,Y 502.823,Z 225.853,A -85,B 0,C 180,E1 -5730.714,E2 -5730.714} C_VEL
LIN {X 0,Y 502.863,Z 225.848,A -85,B 0,C 180,E1 -5733.441,E2 -5733.441} C_VEL
LIN {X 0,Y 502.776,Z 225.86,A -85,B 0,C 180,E1 -5736.087,E2 -5736.087} C_VEL
LIN {X 0,Y 502.785,Z 225.857,A -85,B 0,C 180,E1 -5738.691,E2 -5738.691} C_VEL
LIN {X 0,Y 502.832,Z 225.851,A -85,B 0,C 180,E1 -5741.25,E2 -5741.25} C_VEL
LIN {X 0,Y 502.822,Z 225.854,A -85,B 0,C 180,E1 -5743.769,E2 -5743.769} C_VEL
LIN {X 0,Y 502.835,Z 225.852,A -85,B 0,C 180,E1 -5746.256,E2 -5746.256} C_VEL
LIN {X 0,Y 502.897,Z 225.842,A -85,B 0,C 180,E1 -5748.719,E2 -5748.719} C_VEL
LIN {X 0,Y 502.885,Z 225.847,A -85,B 0,C 180,E1 -5751.968,E2 -5751.968} C_VEL
LIN {X 0,Y 502.942,Z 225.837,A -85,B 0,C 180,E1 -5754.388,E2 -5754.388} C_VEL
LIN {X 0,Y 503.027,Z 225.829,A -85,B 0,C 180,E1 -5757.599,E2 -5757.599} C_VEL
LIN {X 0,Y 503.033,Z 225.828,A -85,B 0,C 180,E1 -5760.001,E2 -5760.001} C_VEL
LIN {X 0,Y 503.026,Z 225.826,A -85,B 0,C 180,E1 -5762.403,E2 -5762.403} C_VEL
LIN {X 0,Y 502.938,Z 225.841,A -85,B 0,C 180,E1 -5765.615,E2 -5765.615} C_VEL
LIN {X 0,Y 502.888,Z 225.845,A -85,B 0,C 180,E1 -5768.035,E2 -5768.035} C_VEL
LIN {X 0,Y 502.885,Z 225.846,A -85,B 0,C 180,E1 -5771.284,E2 -5771.284} C_VEL
LIN {X 0,Y 502.849,Z 225.849,A -85,B 0,C 180,E1 -5774.572,E2 -5774.572} C_VEL
LIN {X 0,Y 502.826,Z 225.853,A -85,B 0,C 180,E1 -5777.909,E2 -5777.909} C_VEL
LIN {X 0,Y 502.839,Z 225.851,A -85,B 0,C 180,E1 -5780.537,E2 -5780.537} C_VEL
LIN {X 0,Y 502.796,Z 225.857,A -85,B 0,C 180,E1 -5783.041,E2 -5783.041} C_VEL
LIN {X 0,Y 502.854,Z 225.849,A -85,B 0,C 180,E1 -5786.557,E2 -5786.557} C_VEL
LIN {X 0,Y 502.832,Z 225.852,A -85,B 0,C 180,E1 -5789.288,E2 -5789.288} C_VEL
LIN {X 0,Y 502.791,Z 225.856,A -85,B 0,C 180,E1 -5792.085,E2 -5792.085} C_VEL
LIN {X 0,Y 502.804,Z 225.855,A -85,B 0,C 180,E1 -5794.966,E2 -5794.966} C_VEL
LIN {X 0,Y 502.801,Z 225.854,A -85,B 0,C 180,E1 -5797.954,E2 -5797.954} C_VEL
LIN {X 0,Y 502.829,Z 225.855,A -85,B 0,C 180,E1 -5801.066,E2 -5801.066} C_VEL
LIN {X 0,Y 502.795,Z 225.857,A -85,B 0,C 180,E1 -5804.53,E2 -5804.53} C_VEL
LIN {X 0,Y 502.804,Z 225.855,A -85,B 0,C 180,E1 -5807.86,E2 -5807.86} C_VEL
LIN {X 0,Y 502.847,Z 226.003,A -85,B 0,C 180,E1 -5810.898,E2 -5810.898} C_VEL
LIN {X 0,Y 503.941,Z 232.503,A -85,B 0,C 180,E1 -5813.604,E2 -5813.604} C_VEL
LIN {X 0,Y 504.024,Z 237.01,A -85,B 0,C 180,E1 -5815.355,E2 -5815.355} C_VEL
LIN {X 0,Y 503.701,Z 245.05,A -85,B 0,C 180,E1 -5818.334,E2 -5818.334} C_VEL
LIN {X 0,Y 503.304,Z 254.262,A -85,B 0,C 180,E1 -5821.609,E2 -5821.609} C_VEL
LIN {X 0,Y 503.039,Z 263.513,A -85,B 0,C 180,E1 -5824.778,E2 -5824.778} C_VEL
LIN {X 0,Y 502.776,Z 272.717,A -85,B 0,C 180,E1 -5827.825,E2 -5827.825} C_VEL
LIN {X 0,Y 502.607,Z 281.929,A -85,B 0,C 180,E1 -5830.815,E2 -5830.815} C_VEL
LIN {X 0,Y 502.443,Z 292.571,A -85,B 0,C 180,E1 -5834.171,E2 -5834.171} C_VEL
LIN {X 0,Y 502.354,Z 297.456,A -85,B 0,C 180,E1 -5835.698,E2 -5835.698} C_VEL
LIN {X 0,Y 504.258,Z 311.009,A -85,B 0,C 180,E1 -5836.075,E2 -5836.075} C_VEL
LIN {X 0,Y 504.483,Z 315.262,A -85,B 0,C 180,E1 -5836.223,E2 -5836.223} C_VEL
LIN {X 0,Y 504.151,Z 328.129,A -85,B 0,C 180,E1 -5836.753,E2 -5836.753} C_VEL
LIN {X 0,Y 503.77,Z 340.585,A -85,B 0,C 180,E1 -5837.453,E2 -5837.453} C_VEL
LIN {X 0,Y 503.412,Z 351.256,A -85,B 0,C 180,E1 -5838.218,E2 -5838.218} C_VEL
LIN {X 0,Y 503.12,Z 361.519,A -85,B 0,C 180,E1 -5839.129,E2 -5839.129} C_VEL
LIN {X 0,Y 502.806,Z 370.749,A -85,B 0,C 180,E1 -5840.14,E2 -5840.14} C_VEL
LIN {X 0,Y 502.515,Z 379.742,A -85,B 0,C 180,E1 -5841.352,E2 -5841.352} C_VEL
LIN {X 0,Y 502.351,Z 386.988,A -85,B 0,C 180,E1 -5842.564,E2 -5842.564} C_VEL
LIN {X 0,Y 502.238,Z 391.879,A -85,B 0,C 180,E1 -5843.572,E2 -5843.572} C_VEL
LIN {X 0,Y 502.18,Z 396.634,A -85,B 0,C 180,E1 -5844.78,E2 -5844.78} C_VEL
LIN {X 0,Y 502.167,Z 400.269,A -85,B 0,C 180,E1 -5845.987,E2 -5845.987} C_VEL
LIN {X 0,Y 502.124,Z 402.14,A -85,B 0,C 180,E1 -5846.79,E2 -5846.79} C_VEL
LIN {X 0,Y 502.122,Z 403.546,A -85,B 0,C 180,E1 -5847.593,E2 -5847.593} C_VEL
LIN {X 0,Y 501.996,Z 405.148,A -85,B 0,C 180,E1 -5849.197,E2 -5849.197} C_VEL
LIN {X 0,Y 501.992,Z 405.361,A -85,B 0,C 180,E1 -5849.999,E2 -5849.999} C_VEL
LIN {X 0,Y 502.037,Z 404.526,A -85,B 0,C 180,E1 -5851.604,E2 -5851.604} C_VEL
LIN {X 0,Y 502.121,Z 403.521,A -85,B 0,C 180,E1 -5852.406,E2 -5852.406} C_VEL
LIN {X 0,Y 502.123,Z 402.106,A -85,B 0,C 180,E1 -5853.209,E2 -5853.209} C_VEL
LIN {X 0,Y 502.106,Z 399.135,A -85,B 0,C 180,E1 -5854.414,E2 -5854.414} C_VEL
LIN {X 0,Y 502.221,Z 395.124,A -85,B 0,C 180,E1 -5855.621,E2 -5855.621} C_VEL
LIN {X 0,Y 502.334,Z 389.054,A -85,B 0,C 180,E1 -5857.011,E2 -5857.011} C_VEL
LIN {X 0,Y 502.46,Z 382.209,A -85,B 0,C 180,E1 -5858.242,E2 -5858.242} C_VEL
LIN {X 0,Y 502.692,Z 373.85,A -85,B 0,C 180,E1 -5859.454,E2 -5859.454} C_VEL
LIN {X 0,Y 502.96,Z 365.285,A -85,B 0,C 180,E1 -5860.465,E2 -5860.465} C_VEL
LIN {X 0,Y 503.365,Z 354.717,A -85,B 0,C 180,E1 -5861.475,E2 -5861.475} C_VEL
LIN {X 0,Y 503.629,Z 343.29,A -85,B 0,C 180,E1 -5862.355,E2 -5862.355} C_VEL
LIN {X 0,Y 503.981,Z 332.822,A -85,B 0,C 180,E1 -5862.994,E2 -5862.994} C_VEL
LIN {X 0,Y 504.319,Z 321.069,A -85,B 0,C 180,E1 -5863.549,E2 -5863.549} C_VEL
LIN {X 0,Y 504.333,Z 311.57,A -85,B 0,C 180,E1 -5863.895,E2 -5863.895} C_VEL
LIN {X 0,Y 502.509,Z 298.623,A -85,B 0,C 180,E1 -5864.27,E2 -5864.27} C_VEL
LIN {X 0,Y 502.349,Z 297.013,A -85,B 0,C 180,E1 -5864.326,E2 -5864.326} C_VEL
LIN {X 0,Y 502.437,Z 288.127,A -85,B 0,C 180,E1 -5867.081,E2 -5867.081} C_VEL
LIN {X 0,Y 502.648,Z 278.783,A -85,B 0,C 180,E1 -5870.032,E2 -5870.032} C_VEL
LIN {X 0,Y 502.8,Z 269.498,A -85,B 0,C 180,E1 -5873.039,E2 -5873.039} C_VEL
LIN {X 0,Y 503.034,Z 260.29,A -85,B 0,C 180,E1 -5876.109,E2 -5876.109} C_VEL
LIN {X 0,Y 503.299,Z 251.28,A -85,B 0,C 180,E1 -5879.257,E2 -5879.257} C_VEL
LIN {X 0,Y 503.652,Z 243.666,A -85,B 0,C 180,E1 -5882.022,E2 -5882.022} C_VEL
LIN {X 0,Y 504.02,Z 236.226,A -85,B 0,C 180,E1 -5884.868,E2 -5884.868} C_VEL
LIN {X 0,Y 504.021,Z 233.336,A -85,B 0,C 180,E1 -5886.026,E2 -5886.026} C_VEL
LIN {X 0,Y 503.119,Z 227.592,A -85,B 0,C 180,E1 -5888.531,E2 -5888.531} C_VEL
LIN {X 0,Y 502.824,Z 225.854,A -85,B 0,C 180,E1 -5889.36,E2 -5889.36} C_VEL
LIN {X 0,Y 502.802,Z 225.858,A -85,B 0,C 180,E1 -5892.198,E2 -5892.198} C_VEL
LIN {X 0,Y 502.784,Z 225.859,A -85,B 0,C 180,E1 -5895.469,E2 -5895.469} C_VEL
LIN {X 0,Y 502.82,Z 225.855,A -85,B 0,C 180,E1 -5898.933,E2 -5898.933} C_VEL
LIN {X 0,Y 502.792,Z 225.859,A -85,B 0,C 180,E1 -5902.045,E2 -5902.045} C_VEL
LIN {X 0,Y 502.807,Z 225.855,A -85,B 0,C 180,E1 -5905.034,E2 -5905.034} C_VEL
LIN {X 0,Y 502.782,Z 225.86,A -85,B 0,C 180,E1 -5907.914,E2 -5907.914} C_VEL
LIN {X 0,Y 502.822,Z 225.853,A -85,B 0,C 180,E1 -5910.711,E2 -5910.711} C_VEL
LIN {X 0,Y 502.86,Z 225.85,A -85,B 0,C 180,E1 -5913.438,E2 -5913.438} C_VEL
LIN {X 0,Y 502.772,Z 225.86,A -85,B 0,C 180,E1 -5916.084,E2 -5916.084} C_VEL
LIN {X 0,Y 502.78,Z 225.857,A -85,B 0,C 180,E1 -5918.688,E2 -5918.688} C_VEL
LIN {X 0,Y 502.827,Z 225.853,A -85,B 0,C 180,E1 -5921.247,E2 -5921.247} C_VEL
LIN {X 0,Y 502.819,Z 225.855,A -85,B 0,C 180,E1 -5923.766,E2 -5923.766} C_VEL
LIN {X 0,Y 502.828,Z 225.853,A -85,B 0,C 180,E1 -5926.254,E2 -5926.254} C_VEL
LIN {X 0,Y 502.888,Z 225.844,A -85,B 0,C 180,E1 -5928.716,E2 -5928.716} C_VEL
LIN {X 0,Y 502.897,Z 225.844,A -85,B 0,C 180,E1 -5931.965,E2 -5931.965} C_VEL
LIN {X 0,Y 502.934,Z 225.838,A -85,B 0,C 180,E1 -5934.385,E2 -5934.385} C_VEL
LIN {X 0,Y 503.019,Z 225.829,A -85,B 0,C 180,E1 -5937.597,E2 -5937.597} C_VEL
LIN {X 0,Y 503.021,Z 225.828,A -85,B 0,C 180,E1 -5939.999,E2 -5939.999} C_VEL
LIN {X 0,Y 503.021,Z 225.828,A -85,B 0,C 180,E1 -5942.401,E2 -5942.401} C_VEL
LIN {X 0,Y 502.933,Z 225.839,A -85,B 0,C 180,E1 -5945.612,E2 -5945.612} C_VEL
LIN {X 0,Y 502.895,Z 225.844,A -85,B 0,C 180,E1 -5948.032,E2 -5948.032} C_VEL
LIN {X 0,Y 502.89,Z 225.845,A -85,B 0,C 180,E1 -5951.281,E2 -5951.281} C_VEL
LIN {X 0,Y 502.837,Z 225.854,A -85,B 0,C 180,E1 -5954.57,E2 -5954.57} C_VEL
LIN {X 0,Y 502.8,Z 225.858,A -85,B 0,C 180,E1 -5957.068,E2 -5957.068} C_VEL
LIN {X 0,Y 502.529,Z 225.893,A -85,B 0,C 180,E1 -5959.61,E2 -5959.61} C_VEL
LIN {X 0,Y 502.472,Z 228.431,A -85,B 0,C 180,E1 -5962.186,E2 -5962.186} C_VEL
LIN {X 0,Y 502.46,Z 231.225,A -85,B 0,C 180,E1 -5964.809,E2 -5964.809} C_VEL
LIN {X 0,Y 502.373,Z 234.857,A -85,B 0,C 180,E1 -5968.197,E2 -5968.197} C_VEL
LIN {X 0,Y 502.272,Z 238.342,A -85,B 0,C 180,E1 -5971.403,E2 -5971.403} C_VEL
LIN {X 0,Y 502.201,Z 241.563,A -85,B 0,C 180,E1 -5974.345,E2 -5974.345} C_VEL
LIN {X 0,Y 502.133,Z 244.615,A -85,B 0,C 180,E1 -5977.082,E2 -5977.082} C_VEL
LIN {X 0,Y 502.176,Z 246.581,A -85,B 0,C 180,E1 -5978.814,E2 -5978.814} C_VEL
LIN {X 0,Y 504.672,Z 258.129,A -85,B 0,C 180,E1 -5979.204,E2 -5979.204} C_VEL
LIN {X 0,Y 504.492,Z 270.832,A -85,B 0,C 180,E1 -5979.707,E2 -5979.707} C_VEL
LIN {X 0,Y 504.168,Z 282.925,A -85,B 0,C 180,E1 -5980.354,E2 -5980.354} C_VEL
LIN {X 0,Y 503.79,Z 293.988,A -85,B 0,C 180,E1 -5981.123,E2 -5981.123} C_VEL
LIN {X 0,Y 503.453,Z 304.826,A -85,B 0,C 180,E1 -5982.069,E2 -5982.069} C_VEL
LIN {X 0,Y 503.139,Z 313.643,A -85,B 0,C 180,E1 -5983.016,E2 -5983.016} C_VEL
LIN {X 0,Y 502.842,Z 322.269,A -85,B 0,C 180,E1 -5984.155,E2 -5984.155} C_VEL
LIN {X 0,Y 502.546,Z 330.382,A -85,B 0,C 180,E1 -5985.495,E2 -5985.495} C_VEL
LIN {X 0,Y 502.38,Z 336.284,A -85,B 0,C 180,E1 -5986.728,E2 -5986.728} C_VEL
LIN {X 0,Y 502.256,Z 340.59,A -85,B 0,C 180,E1 -5987.867,E2 -5987.867} C_VEL
LIN {X 0,Y 502.18,Z 344.137,A -85,B 0,C 180,E1 -5989.086,E2 -5989.086} C_VEL
LIN {X 0,Y 502.065,Z 346.895,A -85,B 0,C 180,E1 -5990.453,E2 -5990.453} C_VEL
LIN {X 0,Y 501.346,Z 347.884,A -85,B 0,C 180,E1 -5991.115,E2 -5991.115} C_VEL
LIN {X 0,Y 498.418,Z 348.934,A -85,B 0,C 180,E1 -5992.195,E2 -5992.195} C_VEL
LIN {X 0,Y 495.534,Z 349.298,A -85,B 0,C 180,E1 -5993.292,E2 -5993.292} C_VEL
LIN {X 0,Y 494.895,Z 349.061,A -85,B 0,C 180,E1 -5993.974,E2 -5993.974} C_VEL
LIN {X 0,Y 494.981,Z 347.616,A -85,B 0,C 180,E1 -5995.435,E2 -5995.435} C_VEL
LIN {X 0,Y 495.078,Z 344.909,A -85,B 0,C 180,E1 -5996.879,E2 -5996.879} C_VEL
LIN {X 0,Y 495.218,Z 340.635,A -85,B 0,C 180,E1 -5998.372,E2 -5998.372} C_VEL
LIN {X 0,Y 495.343,Z 335.742,A -85,B 0,C 180,E1 -5999.64,E2 -5999.64} C_VEL
LIN {X 0,Y 495.542,Z 329.351,A -85,B 0,C 180,E1 -6000.939,E2 -6000.939} C_VEL
LIN {X 0,Y 495.833,Z 322.153,A -85,B 0,C 180,E1 -6002.113,E2 -6002.113} C_VEL
LIN {X 0,Y 496.134,Z 313.443,A -85,B 0,C 180,E1 -6003.262,E2 -6003.262} C_VEL
LIN {X 0,Y 496.553,Z 303.557,A -85,B 0,C 180,E1 -6004.314,E2 -6004.314} C_VEL
LIN {X 0,Y 496.91,Z 292.94,A -85,B 0,C 180,E1 -6005.23,E2 -6005.23} C_VEL
LIN {X 0,Y 497.298,Z 280.777,A -85,B 0,C 180,E1 -6006.05,E2 -6006.05} C_VEL
LIN {X 0,Y 497.619,Z 267.997,A -85,B 0,C 180,E1 -6006.707,E2 -6006.707} C_VEL
LIN {X 0,Y 497.715,Z 258.655,A -85,B 0,C 180,E1 -6007.067,E2 -6007.067} C_VEL
LIN {X 0,Y 495.126,Z 246.481,A -85,B 0,C 180,E1 -6007.493,E2 -6007.493} C_VEL
LIN {X 0,Y 495.144,Z 243.54,A -85,B 0,C 180,E1 -6010.084,E2 -6010.084} C_VEL
LIN {X 0,Y 495.172,Z 240.634,A -85,B 0,C 180,E1 -6012.66,E2 -6012.66} C_VEL
LIN {X 0,Y 495.241,Z 237.792,A -85,B 0,C 180,E1 -6015.201,E2 -6015.201} C_VEL
LIN {X 0,Y 495.311,Z 234.09,A -85,B 0,C 180,E1 -6018.543,E2 -6018.543} C_VEL
LIN {X 0,Y 495.366,Z 230.475,A -85,B 0,C 180,E1 -6021.844,E2 -6021.844} C_VEL
LIN {X 0,Y 495.363,Z 227.791,A -85,B 0,C 180,E1 -6024.301,E2 -6024.301} C_VEL
LIN {X 0,Y 495.429,Z 226.901,A -85,B 0,C 180,E1 -6025.118,E2 -6025.118} C_VEL
LIN {X 0,Y 495.834,Z 226.723,A -85,B 0,C 180,E1 -6028.376,E2 -6028.376} C_VEL
LIN {X 0,Y 495.982,Z 226.704,A -85,B 0,C 180,E1 -6030.001,E2 -6030.001} C_VEL
LIN {X 0,Y 495.98,Z 226.703,A -85,B 0,C 180,E1 -6032.437,E2 -6032.437} C_VEL
LIN {X 0,Y 495.883,Z 226.717,A -85,B 0,C 180,E1 -6035.694,E2 -6035.694} C_VEL
LIN {X 0,Y 495.86,Z 226.719,A -85,B 0,C 180,E1 -6038.149,E2 -6038.149} C_VEL
LIN {X 0,Y 495.864,Z 226.72,A -85,B 0,C 180,E1 -6041.446,E2 -6041.446} C_VEL
LIN {X 0,Y 495.777,Z 226.731,A -85,B 0,C 180,E1 -6044.784,E2 -6044.784} C_VEL
LIN {X 0,Y 495.776,Z 226.731,A -85,B 0,C 180,E1 -6047.32,E2 -6047.32} C_VEL
LIN {X 0,Y 495.766,Z 226.732,A -85,B 0,C 180,E1 -6049.891,E2 -6049.891} C_VEL
LIN {X 0,Y 495.753,Z 226.734,A -85,B 0,C 180,E1 -6052.864,E2 -6052.864} C_VEL
LIN {X 0,Y 495.789,Z 226.729,A -85,B 0,C 180,E1 -6056.069,E2 -6056.069} C_VEL
LIN {X 0,Y 495.762,Z 226.733,A -85,B 0,C 180,E1 -6058.816,E2 -6058.816} C_VEL
LIN {X 0,Y 495.749,Z 226.733,A -85,B 0,C 180,E1 -6061.728,E2 -6061.728} C_VEL
LIN {X 0,Y 495.769,Z 226.732,A -85,B 0,C 180,E1 -6064.697,E2 -6064.697} C_VEL
LIN {X 0,Y 495.724,Z 226.736,A -85,B 0,C 180,E1 -6067.563,E2 -6067.563} C_VEL
LIN {X 0,Y 495.773,Z 226.733,A -85,B 0,C 180,E1 -6070.7,E2 -6070.7} C_VEL
LIN {X 0,Y 495.729,Z 226.735,A -85,B 0,C 180,E1 -6073.697,E2 -6073.697} C_VEL
LIN {X 0,Y 495.723,Z 226.738,A -85,B 0,C 180,E1 -6076.307,E2 -6076.307} C_VEL
LIN {X 0,Y 495.777,Z 226.729,A -85,B 0,C 180,E1 -6079.303,E2 -6079.303} C_VEL
LIN {X 0,Y 495.76,Z 226.731,A -85,B 0,C 180,E1 -6081.412,E2 -6081.412} C_VEL
LIN {X 0,Y 495.753,Z 226.735,A -85,B 0,C 180,E1 -6084.465,E2 -6084.465} C_VEL
LIN {X 0,Y 495.766,Z 226.73,A -85,B 0,C 180,E1 -6087.408,E2 -6087.408} C_VEL
LIN {X 0,Y 495.765,Z 226.733,A -85,B 0,C 180,E1 -6090.255,E2 -6090.255} C_VEL
LIN {X 0,Y 495.824,Z 226.724,A -85,B 0,C 180,E1 -6093.253,E2 -6093.253} C_VEL
LIN {X 0,Y 495.744,Z 226.735,A -85,B 0,C 180,E1 -6096.614,E2 -6096.614} C_VEL
LIN {X 0,Y 495.78,Z 226.73,A -85,B 0,C 180,E1 -6099.326,E2 -6099.326} C_VEL
LIN {X 0,Y 495.796,Z 226.729,A -85,B 0,C 180,E1 -6101.831,E2 -6101.831} C_VEL
LIN {X 0,Y 495.827,Z 226.724,A -85,B 0,C 180,E1 -6104.55,E2 -6104.55} C_VEL
LIN {X 0,Y 495.881,Z 226.718,A -85,B 0,C 180,E1 -6107.941,E2 -6107.941} C_VEL
LIN {X 0,Y 495.839,Z 226.723,A -85,B 0,C 180,E1 -6111.032,E2 -6111.032} C_VEL
LIN {X 0,Y 495.885,Z 226.717,A -85,B 0,C 180,E1 -6113.491,E2 -6113.491} C_VEL
LIN {X 0,Y 495.844,Z 226.721,A -85,B 0,C 180,E1 -6116.751,E2 -6116.751} C_VEL
LIN {X 0,Y 495.876,Z 226.719,A -85,B 0,C 180,E1 -6118.377,E2 -6118.377} C_VEL
LIN {X 0,Y 495.989,Z 226.704,A -85,B 0,C 180,E1 -6120.813,E2 -6120.813} C_VEL
LIN {X 0,Y 495.994,Z 226.702,A -85,B 0,C 180,E1 -6122.438,E2 -6122.438} C_VEL
LIN {X 0,Y 495.894,Z 226.718,A -85,B 0,C 180,E1 -6125.695,E2 -6125.695} C_VEL
LIN {X 0,Y 495.844,Z 226.721,A -85,B 0,C 180,E1 -6128.15,E2 -6128.15} C_VEL
LIN {X 0,Y 495.86,Z 226.722,A -85,B 0,C 180,E1 -6131.446,E2 -6131.446} C_VEL
LIN {X 0,Y 495.796,Z 226.728,A -85,B 0,C 180,E1 -6134.784,E2 -6134.784} C_VEL
LIN {X 0,Y 495.766,Z 226.733,A -85,B 0,C 180,E1 -6137.32,E2 -6137.32} C_VEL
LIN {X 0,Y 495.777,Z 226.73,A -85,B 0,C 180,E1 -6139.891,E2 -6139.891} C_VEL
LIN {X 0,Y 495.767,Z 226.733,A -85,B 0,C 180,E1 -6142.861,E2 -6142.861} C_VEL
LIN {X 0,Y 495.764,Z 226.732,A -85,B 0,C 180,E1 -6146.07,E2 -6146.07} C_VEL
LIN {X 0,Y 495.78,Z 226.731,A -85,B 0,C 180,E1 -6148.815,E2 -6148.815} C_VEL
LIN {X 0,Y 495.763,Z 226.734,A -85,B 0,C 180,E1 -6151.725,E2 -6151.725} C_VEL
LIN {X 0,Y 495.771,Z 226.731,A -85,B 0,C 180,E1 -6154.693,E2 -6154.693} C_VEL
LIN {X 0,Y 495.738,Z 226.737,A -85,B 0,C 180,E1 -6157.562,E2 -6157.562} C_VEL
LIN {X 0,Y 495.775,Z 226.731,A -85,B 0,C 180,E1 -6160.7,E2 -6160.7} C_VEL
LIN {X 0,Y 495.737,Z 226.735,A -85,B 0,C 180,E1 -6164.002,E2 -6164.002} C_VEL
LIN {X 0,Y 495.734,Z 226.734,A -85,B 0,C 180,E1 -6167.117,E2 -6167.117} C_VEL
LIN {X 0,Y 495.767,Z 226.733,A -85,B 0,C 180,E1 -6169.953,E2 -6169.953} C_VEL
LIN {X 0,Y 495.758,Z 226.742,A -85,B 0,C 180,E1 -6170.587,E2 -6170.587} C_VEL
LIN {X 0,Y 496.806,Z 232.505,A -85,B 0,C 180,E1 -6173.042,E2 -6173.042} C_VEL
LIN {X 0,Y 497.118,Z 236.318,A -85,B 0,C 180,E1 -6174.574,E2 -6174.574} C_VEL
LIN {X 0,Y 496.793,Z 243.935,A -85,B 0,C 180,E1 -6177.48,E2 -6177.48} C_VEL
LIN {X 0,Y 496.386,Z 252.915,A -85,B 0,C 180,E1 -6180.76,E2 -6180.76} C_VEL
LIN {X 0,Y 496.067,Z 261.997,A -85,B 0,C 180,E1 -6183.947,E2 -6183.947} C_VEL
LIN {X 0,Y 495.795,Z 271.345,A -85,B 0,C 180,E1 -6187.131,E2 -6187.131} C_VEL
LIN {X 0,Y 495.547,Z 281.65,A -85,B 0,C 180,E1 -6190.531,E2 -6190.531} C_VEL
LIN {X 0,Y 495.383,Z 292.189,A -85,B 0,C 180,E1 -6193.939,E2 -6193.939} C_VEL
LIN {X 0,Y 495.275,Z 297.07,A -85,B 0,C 180,E1 -6195.489,E2 -6195.489} C_VEL
LIN {X 0,Y 497.219,Z 311.005,A -85,B 0,C 180,E1 -6195.887,E2 -6195.887} C_VEL
LIN {X 0,Y 497.543,Z 315.598,A -85,B 0,C 180,E1 -6196.053,E2 -6196.053} C_VEL
LIN {X 0,Y 497.219,Z 327.716,A -85,B 0,C 180,E1 -6196.564,E2 -6196.564} C_VEL
LIN {X 0,Y 496.835,Z 339.293,A -85,B 0,C 180,E1 -6197.218,E2 -6197.218} C_VEL
LIN {X 0,Y 496.396,Z 350.845,A -85,B 0,C 180,E1 -6198.049,E2 -6198.049} C_VEL
LIN {X 0,Y 496.129,Z 361.115,A -85,B 0,C 180,E1 -6198.974,E2 -6198.974} C_VEL
LIN {X 0,Y 495.755,Z 370.345,A -85,B 0,C 180,E1 -6199.998,E2 -6199.998} C_VEL
LIN {X 0,Y 495.453,Z 379.34,A -85,B 0,C 180,E1 -6201.228,E2 -6201.228} C_VEL
LIN {X 0,Y 495.282,Z 386.589,A -85,B 0,C 180,E1 -6202.457,E2 -6202.457} C_VEL
LIN {X 0,Y 495.124,Z 392.686,A -85,B 0,C 180,E1 -6203.761,E2 -6203.761} C_VEL
LIN {X 0,Y 495.038,Z 397.559,A -85,B 0,C 180,E1 -6205.113,E2 -6205.113} C_VEL
LIN {X 0,Y 495.058,Z 399.872,A -85,B 0,C 180,E1 -6205.929,E2 -6205.929} C_VEL
LIN {X 0,Y 495.046,Z 401.745,A -85,B 0,C 180,E1 -6206.744,E2 -6206.744} C_VEL
LIN {X 0,Y 495.055,Z 403.151,A -85,B 0,C 180,E1 -6207.558,E2 -6207.558} C_VEL
LIN {X 0,Y 494.916,Z 404.751,A -85,B 0,C 180,E1 -6209.186,E2 -6209.186} C_VEL
LIN {X 0,Y 494.909,Z 404.964,A -85,B 0,C 180,E1 -6209.999,E2 -6209.999} C_VEL
LIN {X 0,Y 494.964,Z 404.125,A -85,B 0,C 180,E1 -6211.626,E2 -6211.626} C_VEL
LIN {X 0,Y 495.054,Z 403.118,A -85,B 0,C 180,E1 -6212.44,E2 -6212.44} C_VEL
LIN {X 0,Y 495.046,Z 401.702,A -85,B 0,C 180,E1 -6213.255,E2 -6213.255} C_VEL
LIN {X 0,Y 495.011,Z 398.725,A -85,B 0,C 180,E1 -6214.478,E2 -6214.478} C_VEL
LIN {X 0,Y 495.134,Z 394.709,A -85,B 0,C 180,E1 -6215.701,E2 -6215.701} C_VEL
LIN {X 0,Y 495.258,Z 388.531,A -85,B 0,C 180,E1 -6217.132,E2 -6217.132} C_VEL
LIN {X 0,Y 495.383,Z 381.781,A -85,B 0,C 180,E1 -6218.361,E2 -6218.361} C_VEL
LIN {X 0,Y 495.65,Z 373.417,A -85,B 0,C 180,E1 -6219.59,E2 -6219.59} C_VEL
LIN {X 0,Y 495.957,Z 364.846,A -85,B 0,C 180,E1 -6220.615,E2 -6220.615} C_VEL
LIN {X 0,Y 496.359,Z 354.27,A -85,B 0,C 180,E1 -6221.639,E2 -6221.639} C_VEL
LIN {X 0,Y 496.649,Z 342.806,A -85,B 0,C 180,E1 -6222.534,E2 -6222.534} C_VEL
LIN {X 0,Y 497.085,Z 330.411,A -85,B 0,C 180,E1 -6223.281,E2 -6223.281} C_VEL
LIN {X 0,Y 497.476,Z 318.011,A -85,B 0,C 180,E1 -6223.843,E2 -6223.843} C_VEL
LIN {X 0,Y 497.331,Z 311.864,A -85,B 0,C 180,E1 -6224.069,E2 -6224.069} C_VEL
LIN {X 0,Y 495.559,Z 298.917,A -85,B 0,C 180,E1 -6224.461,E2 -6224.461} C_VEL
LIN {X 0,Y 495.254,Z 296.576,A -85,B 0,C 180,E1 -6224.536,E2 -6224.536} C_VEL
LIN {X 0,Y 495.376,Z 287.744,A -85,B 0,C 180,E1 -6227.332,E2 -6227.332} C_VEL
LIN {X 0,Y 495.596,Z 278.666,A -85,B 0,C 180,E1 -6230.259,E2 -6230.259} C_VEL
LIN {X 0,Y 495.753,Z 269.173,A -85,B 0,C 180,E1 -6233.386,E2 -6233.386} C_VEL
LIN {X 0,Y 496.002,Z 260.32,A -85,B 0,C 180,E1 -6236.423,E2 -6236.423} C_VEL
LIN {X 0,Y 496.27,Z 252.372,A -85,B 0,C 180,E1 -6239.246,E2 -6239.246} C_VEL
LIN {X 0,Y 496.63,Z 245.195,A -85,B 0,C 180,E1 -6241.887,E2 -6241.887} C_VEL
LIN {X 0,Y 496.982,Z 238.603,A -85,B 0,C 180,E1 -6244.447,E2 -6244.447} C_VEL
LIN {X 0,Y 496.93,Z 233.738,A -85,B 0,C 180,E1 -6246.44,E2 -6246.44} C_VEL
LIN {X 0,Y 495.921,Z 227.646,A -85,B 0,C 180,E1 -6249.177,E2 -6249.177} C_VEL
LIN {X 0,Y 495.76,Z 226.733,A -85,B 0,C 180,E1 -6249.636,E2 -6249.636} C_VEL
LIN {X 0,Y 495.737,Z 226.736,A -85,B 0,C 180,E1 -6252.506,E2 -6252.506} C_VEL
LIN {X 0,Y 495.736,Z 226.737,A -85,B 0,C 180,E1 -6255.14,E2 -6255.14} C_VEL
LIN {X 0,Y 495.757,Z 226.733,A -85,B 0,C 180,E1 -6258.218,E2 -6258.218} C_VEL
LIN {X 0,Y 495.749,Z 226.735,A -85,B 0,C 180,E1 -6261.407,E2 -6261.407} C_VEL
LIN {X 0,Y 495.754,Z 226.736,A -85,B 0,C 180,E1 -6264.462,E2 -6264.462} C_VEL
LIN {X 0,Y 495.766,Z 226.732,A -85,B 0,C 180,E1 -6267.405,E2 -6267.405} C_VEL
LIN {X 0,Y 495.764,Z 226.734,A -85,B 0,C 180,E1 -6270.253,E2 -6270.253} C_VEL
LIN {X 0,Y 495.821,Z 226.726,A -85,B 0,C 180,E1 -6273.25,E2 -6273.25} C_VEL
LIN {X 0,Y 495.739,Z 226.735,A -85,B 0,C 180,E1 -6276.611,E2 -6276.611} C_VEL
LIN {X 0,Y 495.775,Z 226.732,A -85,B 0,C 180,E1 -6279.323,E2 -6279.323} C_VEL
LIN {X 0,Y 495.794,Z 226.728,A -85,B 0,C 180,E1 -6281.828,E2 -6281.828} C_VEL
LIN {X 0,Y 495.82,Z 226.725,A -85,B 0,C 180,E1 -6284.547,E2 -6284.547} C_VEL
LIN {X 0,Y 495.872,Z 226.719,A -85,B 0,C 180,E1 -6287.938,E2 -6287.938} C_VEL
LIN {X 0,Y 495.839,Z 226.723,A -85,B 0,C 180,E1 -6291.029,E2 -6291.029} C_VEL
LIN {X 0,Y 495.876,Z 226.718,A -85,B 0,C 180,E1 -6293.488,E2 -6293.488} C_VEL
LIN {X 0,Y 495.841,Z 226.722,A -85,B 0,C 180,E1 -6296.749,E2 -6296.749} C_VEL
LIN {X 0,Y 495.999,Z 226.703,A -85,B 0,C 180,E1 -6299.187,E2 -6299.187} C_VEL
LIN {X 0,Y 495.864,Z 226.72,A -85,B 0,C 180,E1 -6301.623,E2 -6301.623} C_VEL
LIN {X 0,Y 495.839,Z 226.723,A -85,B 0,C 180,E1 -6303.249,E2 -6303.249} C_VEL
LIN {X 0,Y 495.872,Z 226.719,A -85,B 0,C 180,E1 -6306.509,E2 -6306.509} C_VEL
LIN {X 0,Y 495.839,Z 226.723,A -85,B 0,C 180,E1 -6308.968,E2 -6308.968} C_VEL
LIN {X 0,Y 495.844,Z 226.724,A -85,B 0,C 180,E1 -6312.274,E2 -6312.274} C_VEL
LIN {X 0,Y 495.797,Z 226.732,A -85,B 0,C 180,E1 -6315.623,E2 -6315.623} C_VEL
LIN {X 0,Y 495.679,Z 226.745,A -85,B 0,C 180,E1 -6318.205,E2 -6318.205} C_VEL
LIN {X 0,Y 495.466,Z 226.797,A -85,B 0,C 180,E1 -6319.902,E2 -6319.902} C_VEL
LIN {X 0,Y 495.403,Z 229.83,A -85,B 0,C 180,E1 -6322.765,E2 -6322.765} C_VEL
LIN {X 0,Y 495.36,Z 232.355,A -85,B 0,C 180,E1 -6325.189,E2 -6325.189} C_VEL
LIN {X 0,Y 495.321,Z 235.827,A -85,B 0,C 180,E1 -6328.395,E2 -6328.395} C_VEL
LIN {X 0,Y 495.216,Z 239.351,A -85,B 0,C 180,E1 -6331.673,E2 -6331.673} C_VEL
LIN {X 0,Y 495.147,Z 242.527,A -85,B 0,C 180,E1 -6334.591,E2 -6334.591} C_VEL
LIN {X 0,Y 495.063,Z 245.865,A -85,B 0,C 180,E1 -6337.619,E2 -6337.619} C_VEL
LIN {X 0,Y 495.112,Z 247.104,A -85,B 0,C 180,E1 -6338.609,E2 -6338.609} C_VEL
LIN {X 0,Y 497.798,Z 258.96,A -85,B 0,C 180,E1 -6339.024,E2 -6339.024} C_VEL
LIN {X 0,Y 497.607,Z 271.358,A -85,B 0,C 180,E1 -6339.525,E2 -6339.525} C_VEL
LIN {X 0,Y 497.268,Z 283.071,A -85,B 0,C 180,E1 -6340.159,E2 -6340.159} C_VEL
LIN {X 0,Y 496.842,Z 294.858,A -85,B 0,C 180,E1 -6340.992,E2 -6340.992} C_VEL
LIN {X 0,Y 496.477,Z 305.871,A -85,B 0,C 180,E1 -6341.977,E2 -6341.977} C_VEL
LIN {X 0,Y 496.135,Z 314.99,A -85,B 0,C 180,E1 -6342.99,E2 -6342.99} C_VEL
LIN {X 0,Y 495.773,Z 323.797,A -85,B 0,C 180,E1 -6344.2,E2 -6344.2} C_VEL
LIN {X 0,Y 495.486,Z 331.707,A -85,B 0,C 180,E1 -6345.562,E2 -6345.562} C_VEL
LIN {X 0,Y 495.334,Z 337.003,A -85,B 0,C 180,E1 -6346.713,E2 -6346.713} C_VEL
LIN {X 0,Y 495.177,Z 342.142,A -85,B 0,C 180,E1 -6348.16,E2 -6348.16} C_VEL
LIN {X 0,Y 495.082,Z 345.031,A -85,B 0,C 180,E1 -6349.233,E2 -6349.233} C_VEL
LIN {X 0,Y 494.999,Z 347.301,A -85,B 0,C 180,E1 -6350.435,E2 -6350.435} C_VEL
LIN {X 0,Y 494.953,Z 348.496,A -85,B 0,C 180,E1 -6351.346,E2 -6351.346} C_VEL
LIN {X 0,Y 494.904,Z 349.3,A -85,B 0,C 180,E1 -6352.675,E2 -6352.675} C_VEL
LIN {X 0,Y 494.895,Z 349.061,A -85,B 0,C 180,E1 -6353.974,E2 -6353.974} C_VEL
LIN {X 0,Y 494.269,Z 348.662,A -85,B 0,C 180,E1 -6354.652,E2 -6354.652} C_VEL
LIN {X 0,Y 491.467,Z 347.453,A -85,B 0,C 180,E1 -6355.749,E2 -6355.749} C_VEL
LIN {X 0,Y 489.097,Z 345.928,A -85,B 0,C 180,E1 -6356.622,E2 -6356.622} C_VEL
LIN {X 0,Y 488.098,Z 344.421,A -85,B 0,C 180,E1 -6357.285,E2 -6357.285} C_VEL
LIN {X 0,Y 488.028,Z 343.831,A -85,B 0,C 180,E1 -6357.507,E2 -6357.507} C_VEL
LIN {X 0,Y 488.174,Z 339.874,A -85,B 0,C 180,E1 -6358.785,E2 -6358.785} C_VEL
LIN {X 0,Y 488.395,Z 333.877,A -85,B 0,C 180,E1 -6360.235,E2 -6360.235} C_VEL
LIN {X 0,Y 488.589,Z 328.184,A -85,B 0,C 180,E1 -6361.331,E2 -6361.331} C_VEL
LIN {X 0,Y 488.929,Z 319.921,A -85,B 0,C 180,E1 -6362.615,E2 -6362.615} C_VEL
LIN {X 0,Y 489.286,Z 310.552,A -85,B 0,C 180,E1 -6363.789,E2 -6363.789} C_VEL
LIN {X 0,Y 489.718,Z 300.466,A -85,B 0,C 180,E1 -6364.8,E2 -6364.8} C_VEL
LIN {X 0,Y 490.061,Z 289.976,A -85,B 0,C 180,E1 -6365.651,E2 -6365.651} C_VEL
LIN {X 0,Y 490.497,Z 278.099,A -85,B 0,C 180,E1 -6366.414,E2 -6366.414} C_VEL
LIN {X 0,Y 490.807,Z 266.246,A -85,B 0,C 180,E1 -6366.989,E2 -6366.989} C_VEL
LIN {X 0,Y 490.795,Z 259.338,A -85,B 0,C 180,E1 -6367.256,E2 -6367.256} C_VEL
LIN {X 0,Y 488.052,Z 246.838,A -85,B 0,C 180,E1 -6367.707,E2 -6367.707} C_VEL
LIN {X 0,Y 488.081,Z 243.501,A -85,B 0,C 180,E1 -6370.66,E2 -6370.66} C_VEL
LIN {X 0,Y 488.103,Z 240.583,A -85,B 0,C 180,E1 -6373.264,E2 -6373.264} C_VEL
LIN {X 0,Y 488.15,Z 237.737,A -85,B 0,C 180,E1 -6375.834,E2 -6375.834} C_VEL
LIN {X 0,Y 488.261,Z 234.929,A -85,B 0,C 180,E1 -6378.375,E2 -6378.375} C_VEL
LIN {X 0,Y 488.298,Z 231.28,A -85,B 0,C 180,E1 -6381.726,E2 -6381.726} C_VEL
LIN {X 0,Y 488.303,Z 228.576,A -85,B 0,C 180,E1 -6384.219,E2 -6384.219} C_VEL
LIN {X 0,Y 488.375,Z 227.686,A -85,B 0,C 180,E1 -6385.048,E2 -6385.048} C_VEL
LIN {X 0,Y 488.8,Z 227.599,A -85,B 0,C 180,E1 -6388.353,E2 -6388.353} C_VEL
LIN {X 0,Y 488.963,Z 227.581,A -85,B 0,C 180,E1 -6390.824,E2 -6390.824} C_VEL
LIN {X 0,Y 488.948,Z 227.579,A -85,B 0,C 180,E1 -6392.472,E2 -6392.472} C_VEL
LIN {X 0,Y 488.842,Z 227.594,A -85,B 0,C 180,E1 -6395.777,E2 -6395.777} C_VEL
LIN {X 0,Y 488.805,Z 227.598,A -85,B 0,C 180,E1 -6398.267,E2 -6398.267} C_VEL
LIN {X 0,Y 488.821,Z 227.597,A -85,B 0,C 180,E1 -6401.613,E2 -6401.613} C_VEL
LIN {X 0,Y 488.749,Z 227.606,A -85,B 0,C 180,E1 -6405.002,E2 -6405.002} C_VEL
LIN {X 0,Y 488.742,Z 227.606,A -85,B 0,C 180,E1 -6408.443,E2 -6408.443} C_VEL
LIN {X 0,Y 488.729,Z 227.61,A -85,B 0,C 180,E1 -6411.071,E2 -6411.071} C_VEL
LIN {X 0,Y 488.69,Z 227.612,A -85,B 0,C 180,E1 -6413.746,E2 -6413.746} C_VEL
LIN {X 0,Y 488.788,Z 227.603,A -85,B 0,C 180,E1 -6416.947,E2 -6416.947} C_VEL
LIN {X 0,Y 488.7,Z 227.613,A -85,B 0,C 180,E1 -6420.365,E2 -6420.365} C_VEL
LIN {X 0,Y 488.727,Z 227.609,A -85,B 0,C 180,E1 -6423.486,E2 -6423.486} C_VEL
LIN {X 0,Y 488.681,Z 227.615,A -85,B 0,C 180,E1 -6426.357,E2 -6426.357} C_VEL
LIN {X 0,Y 488.735,Z 227.609,A -85,B 0,C 180,E1 -6429.252,E2 -6429.252} C_VEL
LIN {X 0,Y 488.729,Z 227.609,A -85,B 0,C 180,E1 -6432.523,E2 -6432.523} C_VEL
LIN {X 0,Y 488.706,Z 227.611,A -85,B 0,C 180,E1 -6435.2,E2 -6435.2} C_VEL
LIN {X 0,Y 488.708,Z 227.612,A -85,B 0,C 180,E1 -6438.401,E2 -6438.401} C_VEL
LIN {X 0,Y 488.744,Z 227.607,A -85,B 0,C 180,E1 -6440.943,E2 -6440.943} C_VEL
LIN {X 0,Y 488.681,Z 227.614,A -85,B 0,C 180,E1 -6443.87,E2 -6443.87} C_VEL
LIN {X 0,Y 488.737,Z 227.607,A -85,B 0,C 180,E1 -6446.879,E2 -6446.879} C_VEL
LIN {X 0,Y 488.723,Z 227.608,A -85,B 0,C 180,E1 -6449.783,E2 -6449.783} C_VEL
LIN {X 0,Y 488.792,Z 227.599,A -85,B 0,C 180,E1 -6453.058,E2 -6453.058} C_VEL
LIN {X 0,Y 488.68,Z 227.615,A -85,B 0,C 180,E1 -6456.256,E2 -6456.256} C_VEL
LIN {X 0,Y 488.748,Z 227.606,A -85,B 0,C 180,E1 -6459.177,E2 -6459.177} C_VEL
LIN {X 0,Y 488.762,Z 227.605,A -85,B 0,C 180,E1 -6461.629,E2 -6461.629} C_VEL
LIN {X 0,Y 488.766,Z 227.604,A -85,B 0,C 180,E1 -6465.001,E2 -6465.001} C_VEL
LIN {X 0,Y 488.834,Z 227.596,A -85,B 0,C 180,E1 -6468.39,E2 -6468.39} C_VEL
LIN {X 0,Y 488.79,Z 227.602,A -85,B 0,C 180,E1 -6471.735,E2 -6471.735} C_VEL
LIN {X 0,Y 488.859,Z 227.593,A -85,B 0,C 180,E1 -6474.226,E2 -6474.226} C_VEL
LIN {X 0,Y 488.964,Z 227.58,A -85,B 0,C 180,E1 -6477.53,E2 -6477.53} C_VEL
LIN {X 0,Y 488.941,Z 227.581,A -85,B 0,C 180,E1 -6480.825,E2 -6480.825} C_VEL
LIN {X 0,Y 488.961,Z 227.578,A -85,B 0,C 180,E1 -6482.473,E2 -6482.473} C_VEL
LIN {X 0,Y 488.853,Z 227.594,A -85,B 0,C 180,E1 -6485.777,E2 -6485.777} C_VEL
LIN {X 0,Y 488.793,Z 227.599,A -85,B 0,C 180,E1 -6488.268,E2 -6488.268} C_VEL
LIN {X 0,Y 488.814,Z 227.598,A -85,B 0,C 180,E1 -6491.613,E2 -6491.613} C_VEL
LIN {X 0,Y 488.769,Z 227.605,A -85,B 0,C 180,E1 -6495.001,E2 -6495.001} C_VEL
LIN {X 0,Y 488.754,Z 227.605,A -85,B 0,C 180,E1 -6498.443,E2 -6498.443} C_VEL
LIN {X 0,Y 488.716,Z 227.61,A -85,B 0,C 180,E1 -6501.071,E2 -6501.071} C_VEL
LIN {X 0,Y 488.68,Z 227.616,A -85,B 0,C 180,E1 -6503.747,E2 -6503.747} C_VEL
LIN {X 0,Y 488.757,Z 227.605,A -85,B 0,C 180,E1 -6506.934,E2 -6506.934} C_VEL
LIN {X 0,Y 488.732,Z 227.609,A -85,B 0,C 180,E1 -6509.271,E2 -6509.271} C_VEL
LIN {X 0,Y 488.711,Z 227.61,A -85,B 0,C 180,E1 -6512.147,E2 -6512.147} C_VEL
LIN {X 0,Y 488.724,Z 227.61,A -85,B 0,C 180,E1 -6515.116,E2 -6515.116} C_VEL
LIN {X 0,Y 488.687,Z 227.612,A -85,B 0,C 180,E1 -6518.2,E2 -6518.2} C_VEL
LIN {X 0,Y 488.728,Z 227.608,A -85,B 0,C 180,E1 -6520.345,E2 -6520.345} C_VEL
LIN {X 0,Y 488.693,Z 227.613,A -85,B 0,C 180,E1 -6523.655,E2 -6523.655} C_VEL
LIN {X 0,Y 488.693,Z 227.611,A -85,B 0,C 180,E1 -6526.345,E2 -6526.345} C_VEL
LIN {X 0,Y 488.742,Z 227.607,A -85,B 0,C 180,E1 -6529.676,E2 -6529.676} C_VEL
LIN {X 0,Y 488.748,Z 227.659,A -85,B 0,C 180,E1 -6530.349,E2 -6530.349} C_VEL
LIN {X 0,Y 489.796,Z 233.635,A -85,B 0,C 180,E1 -6532.939,E2 -6532.939} C_VEL
LIN {X 0,Y 490.124,Z 238.24,A -85,B 0,C 180,E1 -6534.82,E2 -6534.82} C_VEL
LIN {X 0,Y 489.796,Z 245.043,A -85,B 0,C 180,E1 -6537.446,E2 -6537.446} C_VEL
LIN {X 0,Y 489.378,Z 254.006,A -85,B 0,C 180,E1 -6540.772,E2 -6540.772} C_VEL
LIN {X 0,Y 489.024,Z 263.055,A -85,B 0,C 180,E1 -6544.002,E2 -6544.002} C_VEL
LIN {X 0,Y 488.729,Z 272.193,A -85,B 0,C 180,E1 -6547.153,E2 -6547.153} C_VEL
LIN {X 0,Y 488.513,Z 281.342,A -85,B 0,C 180,E1 -6550.239,E2 -6550.239} C_VEL
LIN {X 0,Y 488.315,Z 291.855,A -85,B 0,C 180,E1 -6553.7,E2 -6553.7} C_VEL
LIN {X 0,Y 488.201,Z 296.721,A -85,B 0,C 180,E1 -6555.275,E2 -6555.275} C_VEL
LIN {X 0,Y 490.163,Z 310.962,A -85,B 0,C 180,E1 -6555.693,E2 -6555.693} C_VEL
LIN {X 0,Y 490.605,Z 316.593,A -85,B 0,C 180,E1 -6555.904,E2 -6555.904} C_VEL
LIN {X 0,Y 490.268,Z 328.291,A -85,B 0,C 180,E1 -6556.423,E2 -6556.423} C_VEL
LIN {X 0,Y 489.854,Z 339.543,A -85,B 0,C 180,E1 -6557.077,E2 -6557.077} C_VEL
LIN {X 0,Y 489.424,Z 350.436,A -85,B 0,C 180,E1 -6557.876,E2 -6557.876} C_VEL
LIN {X 0,Y 489.07,Z 360.706,A -85,B 0,C 180,E1 -6558.813,E2 -6558.813} C_VEL
LIN {X 0,Y 488.73,Z 369.942,A -85,B 0,C 180,E1 -6559.853,E2 -6559.853} C_VEL
LIN {X 0,Y 488.406,Z 378.939,A -85,B 0,C 180,E1 -6561.1,E2 -6561.1} C_VEL
LIN {X 0,Y 488.214,Z 386.19,A -85,B 0,C 180,E1 -6562.347,E2 -6562.347} C_VEL
LIN {X 0,Y 488.076,Z 391.583,A -85,B 0,C 180,E1 -6563.498,E2 -6563.498} C_VEL
LIN {X 0,Y 488.045,Z 395.843,A -85,B 0,C 180,E1 -6564.628,E2 -6564.628} C_VEL
LIN {X 0,Y 487.953,Z 399.474,A -85,B 0,C 180,E1 -6565.869,E2 -6565.869} C_VEL
LIN {X 0,Y 487.97,Z 401.35,A -85,B 0,C 180,E1 -6566.697,E2 -6566.697} C_VEL
LIN {X 0,Y 487.96,Z 402.755,A -85,B 0,C 180,E1 -6567.523,E2 -6567.523} C_VEL
LIN {X 0,Y 487.839,Z 404.354,A -85,B 0,C 180,E1 -6569.174,E2 -6569.174} C_VEL
LIN {X 0,Y 487.83,Z 404.566,A -85,B 0,C 180,E1 -6569.999,E2 -6569.999} C_VEL
LIN {X 0,Y 487.894,Z 403.724,A -85,B 0,C 180,E1 -6571.65,E2 -6571.65} C_VEL
LIN {X 0,Y 487.96,Z 402.715,A -85,B 0,C 180,E1 -6572.476,E2 -6572.476} C_VEL
LIN {X 0,Y 487.97,Z 401.297,A -85,B 0,C 180,E1 -6573.302,E2 -6573.302} C_VEL
LIN {X 0,Y 487.923,Z 398.316,A -85,B 0,C 180,E1 -6574.543,E2 -6574.543} C_VEL
LIN {X 0,Y 488.028,Z 394.293,A -85,B 0,C 180,E1 -6575.785,E2 -6575.785} C_VEL
LIN {X 0,Y 488.183,Z 388.109,A -85,B 0,C 180,E1 -6577.236,E2 -6577.236} C_VEL
LIN {X 0,Y 488.326,Z 381.354,A -85,B 0,C 180,E1 -6578.482,E2 -6578.482} C_VEL
LIN {X 0,Y 488.58,Z 372.984,A -85,B 0,C 180,E1 -6579.73,E2 -6579.73} C_VEL
LIN {X 0,Y 488.95,Z 364.41,A -85,B 0,C 180,E1 -6580.769,E2 -6580.769} C_VEL
LIN {X 0,Y 489.358,Z 353.849,A -85,B 0,C 180,E1 -6581.807,E2 -6581.807} C_VEL
LIN {X 0,Y 489.703,Z 342.366,A -85,B 0,C 180,E1 -6582.715,E2 -6582.715} C_VEL
LIN {X 0,Y 490.159,Z 329.969,A -85,B 0,C 180,E1 -6583.473,E2 -6583.473} C_VEL
LIN {X 0,Y 490.56,Z 317.57,A -85,B 0,C 180,E1 -6584.042,E2 -6584.042} C_VEL
LIN {X 0,Y 490.432,Z 312.944,A -85,B 0,C 180,E1 -6584.218,E2 -6584.218} C_VEL
LIN {X 0,Y 488.599,Z 299.319,A -85,B 0,C 180,E1 -6584.655,E2 -6584.655} C_VEL
LIN {X 0,Y 488.188,Z 296.159,A -85,B 0,C 180,E1 -6584.751,E2 -6584.751} C_VEL
LIN {X 0,Y 488.304,Z 287.359,A -85,B 0,C 180,E1 -6587.592,E2 -6587.592} C_VEL
LIN {X 0,Y 488.54,Z 277.743,A -85,B 0,C 180,E1 -6590.759,E2 -6590.759} C_VEL
LIN {X 0,Y 488.73,Z 268.887,A -85,B 0,C 180,E1 -6593.743,E2 -6593.743} C_VEL
LIN {X 0,Y 488.95,Z 261.074,A -85,B 0,C 180,E1 -6596.46,E2 -6596.46} C_VEL
LIN {X 0,Y 489.331,Z 252.178,A -85,B 0,C 180,E1 -6599.702,E2 -6599.702} C_VEL
LIN {X 0,Y 489.736,Z 244.655,A -85,B 0,C 180,E1 -6602.556,E2 -6602.556} C_VEL
LIN {X 0,Y 490.072,Z 237.185,A -85,B 0,C 180,E1 -6605.546,E2 -6605.546} C_VEL
LIN {X 0,Y 489.802,Z 233.698,A -85,B 0,C 180,E1 -6607.058,E2 -6607.058} C_VEL
LIN {X 0,Y 488.729,Z 227.61,A -85,B 0,C 180,E1 -6609.919,E2 -6609.919} C_VEL
LIN {X 0,Y 488.709,Z 227.612,A -85,B 0,C 180,E1 -6612.825,E2 -6612.825} C_VEL
LIN {X 0,Y 488.693,Z 227.614,A -85,B 0,C 180,E1 -6615.976,E2 -6615.976} C_VEL
LIN {X 0,Y 488.708,Z 227.613,A -85,B 0,C 180,E1 -6618.583,E2 -6618.583} C_VEL
LIN {X 0,Y 488.703,Z 227.614,A -85,B 0,C 180,E1 -6620.946,E2 -6620.946} C_VEL
LIN {X 0,Y 488.682,Z 227.615,A -85,B 0,C 180,E1 -6623.867,E2 -6623.867} C_VEL
LIN {X 0,Y 488.737,Z 227.609,A -85,B 0,C 180,E1 -6626.876,E2 -6626.876} C_VEL
LIN {X 0,Y 488.721,Z 227.61,A -85,B 0,C 180,E1 -6629.78,E2 -6629.78} C_VEL
LIN {X 0,Y 488.789,Z 227.601,A -85,B 0,C 180,E1 -6633.055,E2 -6633.055} C_VEL
LIN {X 0,Y 488.676,Z 227.615,A -85,B 0,C 180,E1 -6636.253,E2 -6636.253} C_VEL
LIN {X 0,Y 488.743,Z 227.608,A -85,B 0,C 180,E1 -6639.174,E2 -6639.174} C_VEL
LIN {X 0,Y 488.756,Z 227.606,A -85,B 0,C 180,E1 -6641.626,E2 -6641.626} C_VEL
LIN {X 0,Y 488.758,Z 227.606,A -85,B 0,C 180,E1 -6644.998,E2 -6644.998} C_VEL
LIN {X 0,Y 488.825,Z 227.598,A -85,B 0,C 180,E1 -6648.387,E2 -6648.387} C_VEL
LIN {X 0,Y 488.813,Z 227.6,A -85,B 0,C 180,E1 -6651.732,E2 -6651.732} C_VEL
LIN {X 0,Y 488.851,Z 227.593,A -85,B 0,C 180,E1 -6654.223,E2 -6654.223} C_VEL
LIN {X 0,Y 488.956,Z 227.581,A -85,B 0,C 180,E1 -6657.527,E2 -6657.527} C_VEL
LIN {X 0,Y 488.97,Z 227.58,A -85,B 0,C 180,E1 -6660.822,E2 -6660.822} C_VEL
LIN {X 0,Y 488.957,Z 227.58,A -85,B 0,C 180,E1 -6662.47,E2 -6662.47} C_VEL
LIN {X 0,Y 488.849,Z 227.593,A -85,B 0,C 180,E1 -6665.774,E2 -6665.774} C_VEL
LIN {X 0,Y 488.811,Z 227.598,A -85,B 0,C 180,E1 -6668.265,E2 -6668.265} C_VEL
LIN {X 0,Y 488.827,Z 227.596,A -85,B 0,C 180,E1 -6671.61,E2 -6671.61} C_VEL
LIN {X 0,Y 488.753,Z 227.608,A -85,B 0,C 180,E1 -6674.999,E2 -6674.999} C_VEL
LIN {X 0,Y 488.662,Z 227.621,A -85,B 0,C 180,E1 -6677.578,E2 -6677.578} C_VEL
LIN {X 0,Y 488.408,Z 227.922,A -85,B 0,C 180,E1 -6680.202,E2 -6680.202} C_VEL
LIN {X 0,Y 488.352,Z 230.773,A -85,B 0,C 180,E1 -6682.924,E2 -6682.924} C_VEL
LIN {X 0,Y 488.28,Z 233.553,A -85,B 0,C 180,E1 -6685.58,E2 -6685.58} C_VEL
LIN {X 0,Y 488.232,Z 236.714,A -85,B 0,C 180,E1 -6688.59,E2 -6688.59} C_VEL
LIN {X 0,Y 488.145,Z 239.571,A -85,B 0,C 180,E1 -6691.217,E2 -6691.217} C_VEL
LIN {X 0,Y 488.083,Z 242.717,A -85,B 0,C 180,E1 -6694.162,E2 -6694.162} C_VEL
LIN {X 0,Y 487.992,Z 246.074,A -85,B 0,C 180,E1 -6697.218,E2 -6697.218} C_VEL
LIN {X 0,Y 488.016,Z 247.355,A -85,B 0,C 180,E1 -6698.386,E2 -6698.386} C_VEL
LIN {X 0,Y 490.977,Z 260.473,A -85,B 0,C 180,E1 -6698.864,E2 -6698.864} C_VEL
LIN {X 0,Y 490.719,Z 273.199,A -85,B 0,C 180,E1 -6699.4,E2 -6699.4} C_VEL
LIN {X 0,Y 490.328,Z 284.698,A -85,B 0,C 180,E1 -6700.055,E2 -6700.055} C_VEL
LIN {X 0,Y 489.903,Z 295.942,A -85,B 0,C 180,E1 -6700.875,E2 -6700.875} C_VEL
LIN {X 0,Y 489.523,Z 306.519,A -85,B 0,C 180,E1 -6701.842,E2 -6701.842} C_VEL
LIN {X 0,Y 489.152,Z 315.689,A -85,B 0,C 180,E1 -6702.884,E2 -6702.884} C_VEL
LIN {X 0,Y 488.791,Z 323.963,A -85,B 0,C 180,E1 -6704.036,E2 -6704.036} C_VEL
LIN {X 0,Y 488.462,Z 331.856,A -85,B 0,C 180,E1 -6705.403,E2 -6705.403} C_VEL
LIN {X 0,Y 488.248,Z 338.119,A -85,B 0,C 180,E1 -6706.806,E2 -6706.806} C_VEL
LIN {X 0,Y 488.121,Z 342.2,A -85,B 0,C 180,E1 -6707.973,E2 -6707.973} C_VEL
LIN {X 0,Y 488.028,Z 345.173,A -85,B 0,C 180,E1 -6709.064,E2 -6709.064} C_VEL
LIN {X 0,Y 487.954,Z 346.659,A -85,B 0,C 180,E1 -6709.758,E2 -6709.758} C_VEL
LIN {X 0,Y 487.873,Z 348.649,A -85,B 0,C 180,E1 -6711.065,E2 -6711.065} C_VEL
LIN {X 0,Y 487.825,Z 349.648,A -85,B 0,C 180,E1 -6712.405,E2 -6712.405} C_VEL
LIN {X 0,Y 487.82,Z 349.448,A -85,B 0,C 180,E1 -6713.974,E2 -6713.974} C_VEL
LIN {X 0,Y 487.868,Z 348.387,A -85,B 0,C 180,E1 -6715.193,E2 -6715.193} C_VEL
LIN {X 0,Y 488.018,Z 345.537,A -85,B 0,C 180,E1 -6716.823,E2 -6716.823} C_VEL
LIN {X 0,Y 488.028,Z 343.831,A -85,B 0,C 180,E1 -6717.507,E2 -6717.507} C_VEL
LIN {X 0,Y 487.413,Z 342.013,A -85,B 0,C 180,E1 -6718.164,E2 -6718.164} C_VEL
LIN {X 0,Y 484.677,Z 338.657,A -85,B 0,C 180,E1 -6719.218,E2 -6719.218} C_VEL
LIN {X 0,Y 481.977,Z 334.643,A -85,B 0,C 180,E1 -6720.247,E2 -6720.247} C_VEL
LIN {X 0,Y 481.426,Z 331.739,A -85,B 0,C 180,E1 -6720.857,E2 -6720.857} C_VEL
LIN {X 0,Y 481.755,Z 324.209,A -85,B 0,C 180,E1 -6722.173,E2 -6722.173} C_VEL
LIN {X 0,Y 482.124,Z 315.703,A -85,B 0,C 180,E1 -6723.37,E2 -6723.37} C_VEL
LIN {X 0,Y 482.534,Z 307.127,A -85,B 0,C 180,E1 -6724.356,E2 -6724.356} C_VEL
LIN {X 0,Y 482.946,Z 297.461,A -85,B 0,C 180,E1 -6725.269,E2 -6725.269} C_VEL
LIN {X 0,Y 483.299,Z 286.808,A -85,B 0,C 180,E1 -6726.083,E2 -6726.083} C_VEL
LIN {X 0,Y 483.703,Z 274.484,A -85,B 0,C 180,E1 -6726.82,E2 -6726.82} C_VEL
LIN {X 0,Y 484.092,Z 261.945,A -85,B 0,C 180,E1 -6727.374,E2 -6727.374} C_VEL
LIN {X 0,Y 481.827,Z 250.892,A -85,B 0,C 180,E1 -6727.799,E2 -6727.799} C_VEL
LIN {X 0,Y 480.977,Z 247.192,A -85,B 0,C 180,E1 -6727.927,E2 -6727.927} C_VEL
LIN {X 0,Y 481.022,Z 243.451,A -85,B 0,C 180,E1 -6731.251,E2 -6731.251} C_VEL
LIN {X 0,Y 481.122,Z 239.563,A -85,B 0,C 180,E1 -6734.757,E2 -6734.757} C_VEL
LIN {X 0,Y 481.201,Z 235.789,A -85,B 0,C 180,E1 -6738.202,E2 -6738.202} C_VEL
LIN {X 0,Y 481.245,Z 232.111,A -85,B 0,C 180,E1 -6741.603,E2 -6741.603} C_VEL
LIN {X 0,Y 481.244,Z 229.379,A -85,B 0,C 180,E1 -6744.133,E2 -6744.133} C_VEL
LIN {X 0,Y 481.322,Z 228.534,A -85,B 0,C 180,E1 -6744.975,E2 -6744.975} C_VEL
LIN {X 0,Y 481.765,Z 228.475,A -85,B 0,C 180,E1 -6748.329,E2 -6748.329} C_VEL
LIN {X 0,Y 481.913,Z 228.459,A -85,B 0,C 180,E1 -6750.836,E2 -6750.836} C_VEL
LIN {X 0,Y 481.915,Z 228.455,A -85,B 0,C 180,E1 -6752.508,E2 -6752.508} C_VEL
LIN {X 0,Y 481.803,Z 228.471,A -85,B 0,C 180,E1 -6755.861,E2 -6755.861} C_VEL
LIN {X 0,Y 481.751,Z 228.476,A -85,B 0,C 180,E1 -6758.389,E2 -6758.389} C_VEL
LIN {X 0,Y 481.783,Z 228.474,A -85,B 0,C 180,E1 -6761.785,E2 -6761.785} C_VEL
LIN {X 0,Y 481.729,Z 228.481,A -85,B 0,C 180,E1 -6765.225,E2 -6765.225} C_VEL
LIN {X 0,Y 481.7,Z 228.484,A -85,B 0,C 180,E1 -6768.723,E2 -6768.723} C_VEL
LIN {X 0,Y 481.66,Z 228.489,A -85,B 0,C 180,E1 -6771.395,E2 -6771.395} C_VEL
LIN {X 0,Y 481.671,Z 228.486,A -85,B 0,C 180,E1 -6774.114,E2 -6774.114} C_VEL
LIN {X 0,Y 481.741,Z 228.479,A -85,B 0,C 180,E1 -6777.142,E2 -6777.142} C_VEL
LIN {X 0,Y 481.669,Z 228.486,A -85,B 0,C 180,E1 -6779.743,E2 -6779.743} C_VEL
LIN {X 0,Y 481.664,Z 228.491,A -85,B 0,C 180,E1 -6782.676,E2 -6782.676} C_VEL
LIN {X 0,Y 481.635,Z 228.491,A -85,B 0,C 180,E1 -6785.711,E2 -6785.711} C_VEL
LIN {X 0,Y 481.707,Z 228.483,A -85,B 0,C 180,E1 -6789.356,E2 -6789.356} C_VEL
LIN {X 0,Y 481.668,Z 228.488,A -85,B 0,C 180,E1 -6792.16,E2 -6792.16} C_VEL
LIN {X 0,Y 481.654,Z 228.49,A -85,B 0,C 180,E1 -6794.459,E2 -6794.459} C_VEL
LIN {X 0,Y 481.644,Z 228.491,A -85,B 0,C 180,E1 -6797.841,E2 -6797.841} C_VEL
LIN {X 0,Y 481.716,Z 228.483,A -85,B 0,C 180,E1 -6800.647,E2 -6800.647} C_VEL
LIN {X 0,Y 481.639,Z 228.493,A -85,B 0,C 180,E1 -6804.293,E2 -6804.293} C_VEL
LIN {X 0,Y 481.67,Z 228.486,A -85,B 0,C 180,E1 -6807.328,E2 -6807.328} C_VEL
LIN {X 0,Y 481.678,Z 228.488,A -85,B 0,C 180,E1 -6810.261,E2 -6810.261} C_VEL
LIN {X 0,Y 481.745,Z 228.477,A -85,B 0,C 180,E1 -6813.114,E2 -6813.114} C_VEL
LIN {X 0,Y 481.662,Z 228.49,A -85,B 0,C 180,E1 -6815.888,E2 -6815.888} C_VEL
LIN {X 0,Y 481.704,Z 228.483,A -85,B 0,C 180,E1 -6819.029,E2 -6819.029} C_VEL
LIN {X 0,Y 481.707,Z 228.483,A -85,B 0,C 180,E1 -6822.16,E2 -6822.16} C_VEL
LIN {X 0,Y 481.746,Z 228.478,A -85,B 0,C 180,E1 -6824.777,E2 -6824.777} C_VEL
LIN {X 0,Y 481.799,Z 228.473,A -85,B 0,C 180,E1 -6828.218,E2 -6828.218} C_VEL
LIN {X 0,Y 481.744,Z 228.479,A -85,B 0,C 180,E1 -6831.613,E2 -6831.613} C_VEL
LIN {X 0,Y 481.82,Z 228.47,A -85,B 0,C 180,E1 -6834.141,E2 -6834.141} C_VEL
LIN {X 0,Y 481.931,Z 228.456,A -85,B 0,C 180,E1 -6837.494,E2 -6837.494} C_VEL
LIN {X 0,Y 481.892,Z 228.459,A -85,B 0,C 180,E1 -6840.837,E2 -6840.837} C_VEL
LIN {X 0,Y 481.927,Z 228.454,A -85,B 0,C 180,E1 -6842.509,E2 -6842.509} C_VEL
LIN {X 0,Y 481.814,Z 228.47,A -85,B 0,C 180,E1 -6845.862,E2 -6845.862} C_VEL
LIN {X 0,Y 481.747,Z 228.476,A -85,B 0,C 180,E1 -6848.39,E2 -6848.39} C_VEL
LIN {X 0,Y 481.759,Z 228.477,A -85,B 0,C 180,E1 -6851.786,E2 -6851.786} C_VEL
LIN {X 0,Y 481.75,Z 228.478,A -85,B 0,C 180,E1 -6855.225,E2 -6855.225} C_VEL
LIN {X 0,Y 481.716,Z 228.481,A -85,B 0,C 180,E1 -6858.723,E2 -6858.723} C_VEL
LIN {X 0,Y 481.655,Z 228.491,A -85,B 0,C 180,E1 -6861.395,E2 -6861.395} C_VEL
LIN {X 0,Y 481.658,Z 228.488,A -85,B 0,C 180,E1 -6864.115,E2 -6864.115} C_VEL
LIN {X 0,Y 481.725,Z 228.482,A -85,B 0,C 180,E1 -6867.132,E2 -6867.132} C_VEL
LIN {X 0,Y 481.687,Z 228.485,A -85,B 0,C 180,E1 -6869.742,E2 -6869.742} C_VEL
LIN {X 0,Y 481.679,Z 228.486,A -85,B 0,C 180,E1 -6872.675,E2 -6872.675} C_VEL
LIN {X 0,Y 481.645,Z 228.49,A -85,B 0,C 180,E1 -6875.71,E2 -6875.71} C_VEL
LIN {X 0,Y 481.677,Z 228.489,A -85,B 0,C 180,E1 -6878.86,E2 -6878.86} C_VEL
LIN {X 0,Y 481.661,Z 228.489,A -85,B 0,C 180,E1 -6881.913,E2 -6881.913} C_VEL
LIN {X 0,Y 481.664,Z 228.489,A -85,B 0,C 180,E1 -6884.458,E2 -6884.458} C_VEL
LIN {X 0,Y 481.656,Z 228.488,A -85,B 0,C 180,E1 -6887.839,E2 -6887.839} C_VEL
LIN {X 0,Y 481.743,Z 228.657,A -85,B 0,C 180,E1 -6890.145,E2 -6890.145} C_VEL
LIN {X 0,Y 482.98,Z 236.033,A -85,B 0,C 180,E1 -6893.372,E2 -6893.372} C_VEL
LIN {X 0,Y 483.108,Z 239.966,A -85,B 0,C 180,E1 -6894.989,E2 -6894.989} C_VEL
LIN {X 0,Y 482.725,Z 247.689,A -85,B 0,C 180,E1 -6897.997,E2 -6897.997} C_VEL
LIN {X 0,Y 482.277,Z 256.394,A -85,B 0,C 180,E1 -6901.255,E2 -6901.255} C_VEL
LIN {X 0,Y 481.989,Z 264.12,A -85,B 0,C 180,E1 -6904.059,E2 -6904.059} C_VEL
LIN {X 0,Y 481.656,Z 273.211,A -85,B 0,C 180,E1 -6907.252,E2 -6907.252} C_VEL
LIN {X 0,Y 481.422,Z 282.349,A -85,B 0,C 180,E1 -6910.38,E2 -6910.38} C_VEL
LIN {X 0,Y 481.24,Z 292.832,A -85,B 0,C 180,E1 -6913.89,E2 -6913.89} C_VEL
LIN {X 0,Y 481.131,Z 296.354,A -85,B 0,C 180,E1 -6915.053,E2 -6915.053} C_VEL
LIN {X 0,Y 483.068,Z 310.502,A -85,B 0,C 180,E1 -6915.478,E2 -6915.478} C_VEL
LIN {X 0,Y 483.703,Z 316.153,A -85,B 0,C 180,E1 -6915.699,E2 -6915.699} C_VEL
LIN {X 0,Y 483.358,Z 327.86,A -85,B 0,C 180,E1 -6916.225,E2 -6916.225} C_VEL
LIN {X 0,Y 482.916,Z 339.116,A -85,B 0,C 180,E1 -6916.888,E2 -6916.888} C_VEL
LIN {X 0,Y 482.493,Z 349.671,A -85,B 0,C 180,E1 -6917.671,E2 -6917.671} C_VEL
LIN {X 0,Y 482.086,Z 360.292,A -85,B 0,C 180,E1 -6918.649,E2 -6918.649} C_VEL
LIN {X 0,Y 481.711,Z 369.534,A -85,B 0,C 180,E1 -6919.704,E2 -6919.704} C_VEL
LIN {X 0,Y 481.357,Z 378.535,A -85,B 0,C 180,E1 -6920.969,E2 -6920.969} C_VEL
LIN {X 0,Y 481.14,Z 385.789,A -85,B 0,C 180,E1 -6922.234,E2 -6922.234} C_VEL
LIN {X 0,Y 481.003,Z 391.579,A -85,B 0,C 180,E1 -6923.497,E2 -6923.497} C_VEL
LIN {X 0,Y 480.903,Z 396.768,A -85,B 0,C 180,E1 -6924.969,E2 -6924.969} C_VEL
LIN {X 0,Y 480.85,Z 399.077,A -85,B 0,C 180,E1 -6925.808,E2 -6925.808} C_VEL
LIN {X 0,Y 480.895,Z 400.956,A -85,B 0,C 180,E1 -6926.648,E2 -6926.648} C_VEL
LIN {X 0,Y 480.87,Z 402.359,A -85,B 0,C 180,E1 -6927.486,E2 -6927.486} C_VEL
LIN {X 0,Y 480.826,Z 403.355,A -85,B 0,C 180,E1 -6928.324,E2 -6928.324} C_VEL
LIN {X 0,Y 480.753,Z 404.169,A -85,B 0,C 180,E1 -6929.999,E2 -6929.999} C_VEL
LIN {X 0,Y 480.825,Z 403.324,A -85,B 0,C 180,E1 -6931.674,E2 -6931.674} C_VEL
LIN {X 0,Y 480.87,Z 402.311,A -85,B 0,C 180,E1 -6932.512,E2 -6932.512} C_VEL
LIN {X 0,Y 480.895,Z 400.892,A -85,B 0,C 180,E1 -6933.35,E2 -6933.35} C_VEL
LIN {X 0,Y 480.841,Z 397.907,A -85,B 0,C 180,E1 -6934.61,E2 -6934.61} C_VEL
LIN {X 0,Y 480.93,Z 393.88,A -85,B 0,C 180,E1 -6935.87,E2 -6935.87} C_VEL
LIN {X 0,Y 481.108,Z 387.691,A -85,B 0,C 180,E1 -6937.343,E2 -6937.343} C_VEL
LIN {X 0,Y 481.268,Z 380.933,A -85,B 0,C 180,E1 -6938.608,E2 -6938.608} C_VEL
LIN {X 0,Y 481.533,Z 372.557,A -85,B 0,C 180,E1 -6939.874,E2 -6939.874} C_VEL
LIN {X 0,Y 481.925,Z 363.978,A -85,B 0,C 180,E1 -6940.927,E2 -6940.927} C_VEL
LIN {X 0,Y 482.342,Z 353.66,A -85,B 0,C 180,E1 -6941.958,E2 -6941.958} C_VEL
LIN {X 0,Y 482.68,Z 343.221,A -85,B 0,C 180,E1 -6942.807,E2 -6942.807} C_VEL
LIN {X 0,Y 483.152,Z 331.492,A -85,B 0,C 180,E1 -6943.565,E2 -6943.565} C_VEL
LIN {X 0,Y 483.592,Z 319.747,A -85,B 0,C 180,E1 -6944.142,E2 -6944.142} C_VEL
LIN {X 0,Y 483.496,Z 313.674,A -85,B 0,C 180,E1 -6944.386,E2 -6944.386} C_VEL
LIN {X 0,Y 481.63,Z 299.546,A -85,B 0,C 180,E1 -6944.858,E2 -6944.858} C_VEL
LIN {X 0,Y 481.123,Z 295.78,A -85,B 0,C 180,E1 -6944.972,E2 -6944.972} C_VEL
LIN {X 0,Y 481.234,Z 287.004,A -85,B 0,C 180,E1 -6947.859,E2 -6947.859} C_VEL
LIN {X 0,Y 481.485,Z 277.931,A -85,B 0,C 180,E1 -6950.903,E2 -6950.903} C_VEL
LIN {X 0,Y 481.704,Z 268.636,A -85,B 0,C 180,E1 -6954.111,E2 -6954.111} C_VEL
LIN {X 0,Y 481.989,Z 260.003,A -85,B 0,C 180,E1 -6957.194,E2 -6957.194} C_VEL
LIN {X 0,Y 482.373,Z 252.007,A -85,B 0,C 180,E1 -6960.175,E2 -6960.175} C_VEL
LIN {X 0,Y 482.827,Z 244.521,A -85,B 0,C 180,E1 -6963.081,E2 -6963.081} C_VEL
LIN {X 0,Y 483.092,Z 238.441,A -85,B 0,C 180,E1 -6965.584,E2 -6965.584} C_VEL
LIN {X 0,Y 482.913,Z 235.583,A -85,B 0,C 180,E1 -6966.827,E2 -6966.827} C_VEL
LIN {X 0,Y 481.965,Z 230.145,A -85,B 0,C 180,E1 -6969.389,E2 -6969.389} C_VEL
LIN {X 0,Y 481.714,Z 228.483,A -85,B 0,C 180,E1 -6970.262,E2 -6970.262} C_VEL
LIN {X 0,Y 481.638,Z 228.495,A -85,B 0,C 180,E1 -6973.299,E2 -6973.299} C_VEL
LIN {X 0,Y 481.653,Z 228.492,A -85,B 0,C 180,E1 -6975.64,E2 -6975.64} C_VEL
LIN {X 0,Y 481.656,Z 228.491,A -85,B 0,C 180,E1 -6978.957,E2 -6978.957} C_VEL
LIN {X 0,Y 481.654,Z 228.491,A -85,B 0,C 180,E1 -6981.991,E2 -6981.991} C_VEL
LIN {X 0,Y 481.691,Z 228.486,A -85,B 0,C 180,E1 -6985.317,E2 -6985.317} C_VEL
LIN {X 0,Y 481.643,Z 228.491,A -85,B 0,C 180,E1 -6988.31,E2 -6988.31} C_VEL
LIN {X 0,Y 481.698,Z 228.486,A -85,B 0,C 180,E1 -6991.217,E2 -6991.217} C_VEL
LIN {X 0,Y 481.686,Z 228.486,A -85,B 0,C 180,E1 -6994.041,E2 -6994.041} C_VEL
LIN {X 0,Y 481.671,Z 228.489,A -85,B 0,C 180,E1 -6996.811,E2 -6996.811} C_VEL
LIN {X 0,Y 481.694,Z 228.485,A -85,B 0,C 180,E1 -6999.502,E2 -6999.502} C_VEL
LIN {X 0,Y 481.704,Z 228.483,A -85,B 0,C 180,E1 -7002.157,E2 -7002.157} C_VEL
LIN {X 0,Y 481.739,Z 228.48,A -85,B 0,C 180,E1 -7004.775,E2 -7004.775} C_VEL
LIN {X 0,Y 481.791,Z 228.475,A -85,B 0,C 180,E1 -7008.215,E2 -7008.215} C_VEL
LIN {X 0,Y 481.758,Z 228.478,A -85,B 0,C 180,E1 -7011.61,E2 -7011.61} C_VEL
LIN {X 0,Y 481.812,Z 228.471,A -85,B 0,C 180,E1 -7014.138,E2 -7014.138} C_VEL
LIN {X 0,Y 481.923,Z 228.458,A -85,B 0,C 180,E1 -7017.491,E2 -7017.491} C_VEL
LIN {X 0,Y 481.92,Z 228.458,A -85,B 0,C 180,E1 -7020.834,E2 -7020.834} C_VEL
LIN {X 0,Y 481.924,Z 228.456,A -85,B 0,C 180,E1 -7022.506,E2 -7022.506} C_VEL
LIN {X 0,Y 481.81,Z 228.47,A -85,B 0,C 180,E1 -7025.859,E2 -7025.859} C_VEL
LIN {X 0,Y 481.757,Z 228.478,A -85,B 0,C 180,E1 -7028.387,E2 -7028.387} C_VEL
LIN {X 0,Y 481.789,Z 228.473,A -85,B 0,C 180,E1 -7031.782,E2 -7031.782} C_VEL
LIN {X 0,Y 481.733,Z 228.483,A -85,B 0,C 180,E1 -7035.223,E2 -7035.223} C_VEL
LIN {X 0,Y 481.617,Z 228.498,A -85,B 0,C 180,E1 -7037.843,E2 -7037.843} C_VEL
LIN {X 0,Y 481.389,Z 228.526,A -85,B 0,C 180,E1 -7039.619,E2 -7039.619} C_VEL
LIN {X 0,Y 481.373,Z 229.433,A -85,B 0,C 180,E1 -7040.872,E2 -7040.872} C_VEL
LIN {X 0,Y 481.292,Z 232.795,A -85,B 0,C 180,E1 -7044.132,E2 -7044.132} C_VEL
LIN {X 0,Y 481.175,Z 235.824,A -85,B 0,C 180,E1 -7047.008,E2 -7047.008} C_VEL
LIN {X 0,Y 481.118,Z 238.726,A -85,B 0,C 180,E1 -7049.777,E2 -7049.777} C_VEL
LIN {X 0,Y 481.032,Z 241.878,A -85,B 0,C 180,E1 -7052.721,E2 -7052.721} C_VEL
LIN {X 0,Y 480.978,Z 245.164,A -85,B 0,C 180,E1 -7055.764,E2 -7055.764} C_VEL
LIN {X 0,Y 480.973,Z 247.925,A -85,B 0,C 180,E1 -7058.17,E2 -7058.17} C_VEL
LIN {X 0,Y 484.06,Z 261.086,A -85,B 0,C 180,E1 -7058.663,E2 -7058.663} C_VEL
LIN {X 0,Y 483.851,Z 273.261,A -85,B 0,C 180,E1 -7059.184,E2 -7059.184} C_VEL
LIN {X 0,Y 483.427,Z 284.631,A -85,B 0,C 180,E1 -7059.832,E2 -7059.832} C_VEL
LIN {X 0,Y 482.99,Z 295.913,A -85,B 0,C 180,E1 -7060.661,E2 -7060.661} C_VEL
LIN {X 0,Y 482.607,Z 306.351,A -85,B 0,C 180,E1 -7061.621,E2 -7061.621} C_VEL
LIN {X 0,Y 482.155,Z 316.256,A -85,B 0,C 180,E1 -7062.755,E2 -7062.755} C_VEL
LIN {X 0,Y 481.808,Z 323.57,A -85,B 0,C 180,E1 -7063.778,E2 -7063.778} C_VEL
LIN {X 0,Y 481.52,Z 330.673,A -85,B 0,C 180,E1 -7064.989,E2 -7064.989} C_VEL
LIN {X 0,Y 481.25,Z 337.331,A -85,B 0,C 180,E1 -7066.411,E2 -7066.411} C_VEL
LIN {X 0,Y 481.058,Z 342.25,A -85,B 0,C 180,E1 -7067.777,E2 -7067.777} C_VEL
LIN {X 0,Y 480.911,Z 346.536,A -85,B 0,C 180,E1 -7069.455,E2 -7069.455} C_VEL
LIN {X 0,Y 480.805,Z 349.075,A -85,B 0,C 180,E1 -7071.059,E2 -7071.059} C_VEL
LIN {X 0,Y 480.735,Z 349.913,A -85,B 0,C 180,E1 -7072.13,E2 -7072.13} C_VEL
LIN {X 0,Y 480.738,Z 350.069,A -85,B 0,C 180,E1 -7073.516,E2 -7073.516} C_VEL
LIN {X 0,Y 480.777,Z 349.11,A -85,B 0,C 180,E1 -7074.942,E2 -7074.942} C_VEL
LIN {X 0,Y 480.889,Z 346.921,A -85,B 0,C 180,E1 -7076.408,E2 -7076.408} C_VEL
LIN {X 0,Y 480.991,Z 343.239,A -85,B 0,C 180,E1 -7077.933,E2 -7077.933} C_VEL
LIN {X 0,Y 481.165,Z 338.822,A -85,B 0,C 180,E1 -7079.256,E2 -7079.256} C_VEL
LIN {X 0,Y 481.402,Z 332.438,A -85,B 0,C 180,E1 -7080.722,E2 -7080.722} C_VEL
LIN {X 0,Y 481.426,Z 331.739,A -85,B 0,C 180,E1 -7080.857,E2 -7080.857} C_VEL
LIN {X 0,Y 480.888,Z 328.656,A -85,B 0,C 180,E1 -7081.453,E2 -7081.453} C_VEL
LIN {X 0,Y 477.11,Z 321.096,A -85,B 0,C 180,E1 -7082.776,E2 -7082.776} C_VEL
LIN {X 0,Y 475.421,Z 316.193,A -85,B 0,C 180,E1 -7083.496,E2 -7083.496} C_VEL
LIN {X 0,Y 475.236,Z 313.48,A -85,B 0,C 180,E1 -7083.841,E2 -7083.841} C_VEL
LIN {X 0,Y 475.788,Z 302.86,A -85,B 0,C 180,E1 -7084.988,E2 -7084.988} C_VEL
LIN {X 0,Y 476.193,Z 291.97,A -85,B 0,C 180,E1 -7085.922,E2 -7085.922} C_VEL
LIN {X 0,Y 476.621,Z 281.241,A -85,B 0,C 180,E1 -7086.655,E2 -7086.655} C_VEL
LIN {X 0,Y 476.988,Z 269.017,A -85,B 0,C 180,E1 -7087.304,E2 -7087.304} C_VEL
LIN {X 0,Y 477.039,Z 261.359,A -85,B 0,C 180,E1 -7087.621,E2 -7087.621} C_VEL
LIN {X 0,Y 473.898,Z 247.547,A -85,B 0,C 180,E1 -7088.153,E2 -7088.153} C_VEL
LIN {X 0,Y 473.948,Z 243.674,A -85,B 0,C 180,E1 -7091.622,E2 -7091.622} C_VEL
LIN {X 0,Y 474.032,Z 240.468,A -85,B 0,C 180,E1 -7094.523,E2 -7094.523} C_VEL
LIN {X 0,Y 474.119,Z 236.628,A -85,B 0,C 180,E1 -7098.042,E2 -7098.042} C_VEL
LIN {X 0,Y 474.173,Z 232.957,A -85,B 0,C 180,E1 -7101.477,E2 -7101.477} C_VEL
LIN {X 0,Y 474.186,Z 230.191,A -85,B 0,C 180,E1 -7104.046,E2 -7104.046} C_VEL
LIN {X 0,Y 474.271,Z 229.412,A -85,B 0,C 180,E1 -7104.9,E2 -7104.9} C_VEL
LIN {X 0,Y 474.73,Z 229.352,A -85,B 0,C 180,E1 -7108.304,E2 -7108.304} C_VEL
LIN {X 0,Y 474.864,Z 229.337,A -85,B 0,C 180,E1 -7110.849,E2 -7110.849} C_VEL
LIN {X 0,Y 474.881,Z 229.331,A -85,B 0,C 180,E1 -7112.546,E2 -7112.546} C_VEL
LIN {X 0,Y 474.766,Z 229.348,A -85,B 0,C 180,E1 -7115.949,E2 -7115.949} C_VEL
LIN {X 0,Y 474.716,Z 229.353,A -85,B 0,C 180,E1 -7118.515,E2 -7118.515} C_VEL
LIN {X 0,Y 474.726,Z 229.352,A -85,B 0,C 180,E1 -7121.963,E2 -7121.963} C_VEL
LIN {X 0,Y 474.667,Z 229.358,A -85,B 0,C 180,E1 -7125.769,E2 -7125.769} C_VEL
LIN {X 0,Y 474.653,Z 229.363,A -85,B 0,C 180,E1 -7129.012,E2 -7129.012} C_VEL
LIN {X 0,Y 474.597,Z 229.367,A -85,B 0,C 180,E1 -7131.729,E2 -7131.729} C_VEL
LIN {X 0,Y 474.651,Z 229.362,A -85,B 0,C 180,E1 -7134.494,E2 -7134.494} C_VEL
LIN {X 0,Y 474.688,Z 229.357,A -85,B 0,C 180,E1 -7137.34,E2 -7137.34} C_VEL
LIN {X 0,Y 474.595,Z 229.369,A -85,B 0,C 180,E1 -7140.812,E2 -7140.812} C_VEL
LIN {X 0,Y 474.629,Z 229.364,A -85,B 0,C 180,E1 -7143.986,E2 -7143.986} C_VEL
LIN {X 0,Y 474.567,Z 229.373,A -85,B 0,C 180,E1 -7146.902,E2 -7146.902} C_VEL
LIN {X 0,Y 474.643,Z 229.362,A -85,B 0,C 180,E1 -7149.653,E2 -7149.653} C_VEL
LIN {X 0,Y 474.646,Z 229.364,A -85,B 0,C 180,E1 -7152.932,E2 -7152.932} C_VEL
LIN {X 0,Y 474.604,Z 229.367,A -85,B 0,C 180,E1 -7155.897,E2 -7155.897} C_VEL
LIN {X 0,Y 474.637,Z 229.363,A -85,B 0,C 180,E1 -7159.041,E2 -7159.041} C_VEL
LIN {X 0,Y 474.616,Z 229.365,A -85,B 0,C 180,E1 -7161.704,E2 -7161.704} C_VEL
LIN {X 0,Y 474.627,Z 229.365,A -85,B 0,C 180,E1 -7164.728,E2 -7164.728} C_VEL
LIN {X 0,Y 474.634,Z 229.364,A -85,B 0,C 180,E1 -7167.79,E2 -7167.79} C_VEL
LIN {X 0,Y 474.623,Z 229.366,A -85,B 0,C 180,E1 -7170.886,E2 -7170.886} C_VEL
LIN {X 0,Y 474.654,Z 229.362,A -85,B 0,C 180,E1 -7173.63,E2 -7173.63} C_VEL
LIN {X 0,Y 474.636,Z 229.365,A -85,B 0,C 180,E1 -7176.643,E2 -7176.643} C_VEL
LIN {X 0,Y 474.659,Z 229.362,A -85,B 0,C 180,E1 -7180.091,E2 -7180.091} C_VEL
LIN {X 0,Y 474.65,Z 229.361,A -85,B 0,C 180,E1 -7182.776,E2 -7182.776} C_VEL
LIN {X 0,Y 474.652,Z 229.362,A -85,B 0,C 180,E1 -7185.423,E2 -7185.423} C_VEL
LIN {X 0,Y 474.744,Z 229.351,A -85,B 0,C 180,E1 -7188.04,E2 -7188.04} C_VEL
LIN {X 0,Y 474.716,Z 229.353,A -85,B 0,C 180,E1 -7191.488,E2 -7191.488} C_VEL
LIN {X 0,Y 474.783,Z 229.348,A -85,B 0,C 180,E1 -7194.054,E2 -7194.054} C_VEL
LIN {X 0,Y 474.897,Z 229.332,A -85,B 0,C 180,E1 -7197.457,E2 -7197.457} C_VEL
LIN {X 0,Y 474.918,Z 229.329,A -85,B 0,C 180,E1 -7200.001,E2 -7200.001} C_VEL
LIN {X 0,Y 474.893,Z 229.33,A -85,B 0,C 180,E1 -7202.546,E2 -7202.546} C_VEL
LIN {X 0,Y 474.776,Z 229.346,A -85,B 0,C 180,E1 -7205.949,E2 -7205.949} C_VEL
LIN {X 0,Y 474.719,Z 229.352,A -85,B 0,C 180,E1 -7208.515,E2 -7208.515} C_VEL
LIN {X 0,Y 474.713,Z 229.354,A -85,B 0,C 180,E1 -7211.963,E2 -7211.963} C_VEL
LIN {X 0,Y 474.708,Z 229.355,A -85,B 0,C 180,E1 -7215.457,E2 -7215.457} C_VEL
LIN {X 0,Y 474.671,Z 229.359,A -85,B 0,C 180,E1 -7219.011,E2 -7219.011} C_VEL
LIN {X 0,Y 474.598,Z 229.369,A -85,B 0,C 180,E1 -7221.73,E2 -7221.73} C_VEL
LIN {X 0,Y 474.637,Z 229.362,A -85,B 0,C 180,E1 -7224.495,E2 -7224.495} C_VEL
LIN {X 0,Y 474.683,Z 229.36,A -85,B 0,C 180,E1 -7227.333,E2 -7227.333} C_VEL
LIN {X 0,Y 474.613,Z 229.364,A -85,B 0,C 180,E1 -7230.231,E2 -7230.231} C_VEL
LIN {X 0,Y 474.634,Z 229.365,A -85,B 0,C 180,E1 -7233.222,E2 -7233.222} C_VEL
LIN {X 0,Y 474.598,Z 229.368,A -85,B 0,C 180,E1 -7236.324,E2 -7236.324} C_VEL
LIN {X 0,Y 474.625,Z 229.366,A -85,B 0,C 180,E1 -7239.646,E2 -7239.646} C_VEL
LIN {X 0,Y 474.633,Z 229.366,A -85,B 0,C 180,E1 -7242.237,E2 -7242.237} C_VEL
LIN {X 0,Y 474.626,Z 229.364,A -85,B 0,C 180,E1 -7245.298,E2 -7245.298} C_VEL
LIN {X 0,Y 474.629,Z 229.363,A -85,B 0,C 180,E1 -7248.214,E2 -7248.214} C_VEL
LIN {X 0,Y 474.672,Z 229.516,A -85,B 0,C 180,E1 -7249.875,E2 -7249.875} C_VEL
LIN {X 0,Y 475.836,Z 236.261,A -85,B 0,C 180,E1 -7252.9,E2 -7252.9} C_VEL
LIN {X 0,Y 476.163,Z 239.488,A -85,B 0,C 180,E1 -7254.271,E2 -7254.271} C_VEL
LIN {X 0,Y 475.813,Z 247.155,A -85,B 0,C 180,E1 -7257.344,E2 -7257.344} C_VEL
LIN {X 0,Y 475.296,Z 256.161,A -85,B 0,C 180,E1 -7260.793,E2 -7260.793} C_VEL
LIN {X 0,Y 474.945,Z 265.159,A -85,B 0,C 180,E1 -7264.117,E2 -7264.117} C_VEL
LIN {X 0,Y 474.58,Z 274.226,A -85,B 0,C 180,E1 -7267.353,E2 -7267.353} C_VEL
LIN {X 0,Y 474.324,Z 283.349,A -85,B 0,C 180,E1 -7270.525,E2 -7270.525} C_VEL
LIN {X 0,Y 474.126,Z 293.904,A -85,B 0,C 180,E1 -7274.127,E2 -7274.127} C_VEL
LIN {X 0,Y 474.068,Z 296.093,A -85,B 0,C 180,E1 -7274.839,E2 -7274.839} C_VEL
LIN {X 0,Y 475.917,Z 309.575,A -85,B 0,C 180,E1 -7275.241,E2 -7275.241} C_VEL
LIN {X 0,Y 476.776,Z 316.98,A -85,B 0,C 180,E1 -7275.541,E2 -7275.541} C_VEL
LIN {X 0,Y 476.356,Z 329.392,A -85,B 0,C 180,E1 -7276.128,E2 -7276.128} C_VEL
LIN {X 0,Y 475.864,Z 341.355,A -85,B 0,C 180,E1 -7276.874,E2 -7276.874} C_VEL
LIN {X 0,Y 475.395,Z 351.63,A -85,B 0,C 180,E1 -7277.69,E2 -7277.69} C_VEL
LIN {X 0,Y 474.982,Z 361.845,A -85,B 0,C 180,E1 -7278.693,E2 -7278.693} C_VEL
LIN {X 0,Y 474.57,Z 370.758,A -85,B 0,C 180,E1 -7279.763,E2 -7279.763} C_VEL
LIN {X 0,Y 474.237,Z 379.466,A -85,B 0,C 180,E1 -7281.047,E2 -7281.047} C_VEL
LIN {X 0,Y 474.034,Z 386.421,A -85,B 0,C 180,E1 -7282.331,E2 -7282.331} C_VEL
LIN {X 0,Y 473.904,Z 391.658,A -85,B 0,C 180,E1 -7283.525,E2 -7283.525} C_VEL
LIN {X 0,Y 473.836,Z 396.37,A -85,B 0,C 180,E1 -7284.893,E2 -7284.893} C_VEL
LIN {X 0,Y 473.753,Z 398.678,A -85,B 0,C 180,E1 -7285.745,E2 -7285.745} C_VEL
LIN {X 0,Y 473.821,Z 400.558,A -85,B 0,C 180,E1 -7286.598,E2 -7286.598} C_VEL
LIN {X 0,Y 473.784,Z 401.962,A -85,B 0,C 180,E1 -7287.449,E2 -7287.449} C_VEL
LIN {X 0,Y 473.759,Z 402.959,A -85,B 0,C 180,E1 -7288.299,E2 -7288.299} C_VEL
LIN {X 0,Y 473.679,Z 403.771,A -85,B 0,C 180,E1 -7289.999,E2 -7289.999} C_VEL
LIN {X 0,Y 473.759,Z 402.925,A -85,B 0,C 180,E1 -7291.699,E2 -7291.699} C_VEL
LIN {X 0,Y 473.784,Z 401.909,A -85,B 0,C 180,E1 -7292.55,E2 -7292.55} C_VEL
LIN {X 0,Y 473.821,Z 400.489,A -85,B 0,C 180,E1 -7293.401,E2 -7293.401} C_VEL
LIN {X 0,Y 473.765,Z 397.5,A -85,B 0,C 180,E1 -7294.679,E2 -7294.679} C_VEL
LIN {X 0,Y 473.836,Z 393.468,A -85,B 0,C 180,E1 -7295.959,E2 -7295.959} C_VEL
LIN {X 0,Y 474.016,Z 387.273,A -85,B 0,C 180,E1 -7297.453,E2 -7297.453} C_VEL
LIN {X 0,Y 474.18,Z 380.511,A -85,B 0,C 180,E1 -7298.737,E2 -7298.737} C_VEL
LIN {X 0,Y 474.474,Z 372.136,A -85,B 0,C 180,E1 -7300.022,E2 -7300.022} C_VEL
LIN {X 0,Y 474.884,Z 363.558,A -85,B 0,C 180,E1 -7301.092,E2 -7301.092} C_VEL
LIN {X 0,Y 475.326,Z 353.466,A -85,B 0,C 180,E1 -7302.117,E2 -7302.117} C_VEL
LIN {X 0,Y 475.74,Z 342.522,A -85,B 0,C 180,E1 -7303.019,E2 -7303.019} C_VEL
LIN {X 0,Y 476.235,Z 331.088,A -85,B 0,C 180,E1 -7303.765,E2 -7303.765} C_VEL
LIN {X 0,Y 476.693,Z 319.356,A -85,B 0,C 180,E1 -7304.351,E2 -7304.351} C_VEL
LIN {X 0,Y 476.493,Z 314.045,A -85,B 0,C 180,E1 -7304.575,E2 -7304.575} C_VEL
LIN {X 0,Y 474.726,Z 300.209,A -85,B 0,C 180,E1 -7305.055,E2 -7305.055} C_VEL
LIN {X 0,Y 474.046,Z 295.358,A -85,B 0,C 180,E1 -7305.201,E2 -7305.201} C_VEL
LIN {X 0,Y 474.229,Z 285.625,A -85,B 0,C 180,E1 -7308.472,E2 -7308.472} C_VEL
LIN {X 0,Y 474.466,Z 276.156,A -85,B 0,C 180,E1 -7311.734,E2 -7311.734} C_VEL
LIN {X 0,Y 474.741,Z 267.015,A -85,B 0,C 180,E1 -7314.954,E2 -7314.954} C_VEL
LIN {X 0,Y 475.088,Z 258.065,A -85,B 0,C 180,E1 -7318.253,E2 -7318.253} C_VEL
LIN {X 0,Y 475.603,Z 249.344,A -85,B 0,C 180,E1 -7321.639,E2 -7321.639} C_VEL
LIN {X 0,Y 476.028,Z 241.988,A -85,B 0,C 180,E1 -7324.638,E2 -7324.638} C_VEL
LIN {X 0,Y 475.992,Z 237.351,A -85,B 0,C 180,E1 -7326.644,E2 -7326.644} C_VEL
LIN {X 0,Y 474.984,Z 231.345,A -85,B 0,C 180,E1 -7329.511,E2 -7329.511} C_VEL
LIN {X 0,Y 474.64,Z 229.364,A -85,B 0,C 180,E1 -7330.524,E2 -7330.524} C_VEL
LIN {X 0,Y 474.6,Z 229.37,A -85,B 0,C 180,E1 -7333.48,E2 -7333.48} C_VEL
LIN {X 0,Y 474.599,Z 229.371,A -85,B 0,C 180,E1 -7336.518,E2 -7336.518} C_VEL
LIN {X 0,Y 474.616,Z 229.366,A -85,B 0,C 180,E1 -7339.341,E2 -7339.341} C_VEL
LIN {X 0,Y 474.609,Z 229.368,A -85,B 0,C 180,E1 -7341.703,E2 -7341.703} C_VEL
LIN {X 0,Y 474.628,Z 229.366,A -85,B 0,C 180,E1 -7344.725,E2 -7344.725} C_VEL
LIN {X 0,Y 474.634,Z 229.366,A -85,B 0,C 180,E1 -7347.787,E2 -7347.787} C_VEL
LIN {X 0,Y 474.622,Z 229.366,A -85,B 0,C 180,E1 -7350.883,E2 -7350.883} C_VEL
LIN {X 0,Y 474.652,Z 229.364,A -85,B 0,C 180,E1 -7353.627,E2 -7353.627} C_VEL
LIN {X 0,Y 474.631,Z 229.365,A -85,B 0,C 180,E1 -7356.64,E2 -7356.64} C_VEL
LIN {X 0,Y 474.653,Z 229.362,A -85,B 0,C 180,E1 -7360.088,E2 -7360.088} C_VEL
LIN {X 0,Y 474.647,Z 229.363,A -85,B 0,C 180,E1 -7362.773,E2 -7362.773} C_VEL
LIN {X 0,Y 474.644,Z 229.362,A -85,B 0,C 180,E1 -7365.42,E2 -7365.42} C_VEL
LIN {X 0,Y 474.735,Z 229.352,A -85,B 0,C 180,E1 -7368.037,E2 -7368.037} C_VEL
LIN {X 0,Y 474.723,Z 229.354,A -85,B 0,C 180,E1 -7371.485,E2 -7371.485} C_VEL
LIN {X 0,Y 474.775,Z 229.348,A -85,B 0,C 180,E1 -7374.051,E2 -7374.051} C_VEL
LIN {X 0,Y 474.889,Z 229.334,A -85,B 0,C 180,E1 -7377.454,E2 -7377.454} C_VEL
LIN {X 0,Y 474.871,Z 229.336,A -85,B 0,C 180,E1 -7380.847,E2 -7380.847} C_VEL
LIN {X 0,Y 474.89,Z 229.332,A -85,B 0,C 180,E1 -7382.543,E2 -7382.543} C_VEL
LIN {X 0,Y 474.773,Z 229.347,A -85,B 0,C 180,E1 -7385.946,E2 -7385.946} C_VEL
LIN {X 0,Y 474.722,Z 229.355,A -85,B 0,C 180,E1 -7388.512,E2 -7388.512} C_VEL
LIN {X 0,Y 474.731,Z 229.353,A -85,B 0,C 180,E1 -7391.96,E2 -7391.96} C_VEL
LIN {X 0,Y 474.67,Z 229.363,A -85,B 0,C 180,E1 -7395.766,E2 -7395.766} C_VEL
LIN {X 0,Y 474.492,Z 229.384,A -85,B 0,C 180,E1 -7398.572,E2 -7398.572} C_VEL
LIN {X 0,Y 474.306,Z 229.408,A -85,B 0,C 180,E1 -7399.924,E2 -7399.924} C_VEL
LIN {X 0,Y 474.232,Z 232.105,A -85,B 0,C 180,E1 -7402.661,E2 -7402.661} C_VEL
LIN {X 0,Y 474.178,Z 234.927,A -85,B 0,C 180,E1 -7405.454,E2 -7405.454} C_VEL
LIN {X 0,Y 474.09,Z 237.96,A -85,B 0,C 180,E1 -7408.317,E2 -7408.317} C_VEL
LIN {X 0,Y 474.042,Z 241.053,A -85,B 0,C 180,E1 -7411.256,E2 -7411.256} C_VEL
LIN {X 0,Y 473.924,Z 244.28,A -85,B 0,C 180,E1 -7414.297,E2 -7414.297} C_VEL
LIN {X 0,Y 473.874,Z 247.671,A -85,B 0,C 180,E1 -7417.448,E2 -7417.448} C_VEL
LIN {X 0,Y 473.881,Z 248.206,A -85,B 0,C 180,E1 -7417.933,E2 -7417.933} C_VEL
LIN {X 0,Y 477.092,Z 261.699,A -85,B 0,C 180,E1 -7418.452,E2 -7418.452} C_VEL
LIN {X 0,Y 476.953,Z 274.418,A -85,B 0,C 180,E1 -7419.015,E2 -7419.015} C_VEL
LIN {X 0,Y 476.503,Z 286.163,A -85,B 0,C 180,E1 -7419.713,E2 -7419.713} C_VEL
LIN {X 0,Y 476.064,Z 296.671,A -85,B 0,C 180,E1 -7420.506,E2 -7420.506} C_VEL
LIN {X 0,Y 475.648,Z 307.424,A -85,B 0,C 180,E1 -7421.519,E2 -7421.519} C_VEL
LIN {X 0,Y 475.17,Z 316.974,A -85,B 0,C 180,E1 -7422.642,E2 -7422.642} C_VEL
LIN {X 0,Y 474.754,Z 325.228,A -85,B 0,C 180,E1 -7423.838,E2 -7423.838} C_VEL
LIN {X 0,Y 474.465,Z 332.003,A -85,B 0,C 180,E1 -7425.046,E2 -7425.046} C_VEL
LIN {X 0,Y 474.201,Z 337.475,A -85,B 0,C 180,E1 -7426.248,E2 -7426.248} C_VEL
LIN {X 0,Y 474.03,Z 341.886,A -85,B 0,C 180,E1 -7427.46,E2 -7427.46} C_VEL
LIN {X 0,Y 473.912,Z 345.331,A -85,B 0,C 180,E1 -7428.679,E2 -7428.679} C_VEL
LIN {X 0,Y 473.764,Z 348.636,A -85,B 0,C 180,E1 -7430.367,E2 -7430.367} C_VEL
LIN {X 0,Y 473.654,Z 350.167,A -85,B 0,C 180,E1 -7431.848,E2 -7431.848} C_VEL
LIN {X 0,Y 473.659,Z 350.522,A -85,B 0,C 180,E1 -7433.245,E2 -7433.245} C_VEL
LIN {X 0,Y 473.682,Z 349.774,A -85,B 0,C 180,E1 -7434.686,E2 -7434.686} C_VEL
LIN {X 0,Y 473.775,Z 347.816,A -85,B 0,C 180,E1 -7436.168,E2 -7436.168} C_VEL
LIN {X 0,Y 473.9,Z 344.399,A -85,B 0,C 180,E1 -7437.733,E2 -7437.733} C_VEL
LIN {X 0,Y 474.097,Z 339.424,A -85,B 0,C 180,E1 -7439.289,E2 -7439.289} C_VEL
LIN {X 0,Y 474.353,Z 333.304,A -85,B 0,C 180,E1 -7440.731,E2 -7440.731} C_VEL
LIN {X 0,Y 474.677,Z 326.712,A -85,B 0,C 180,E1 -7441.961,E2 -7441.961} C_VEL
LIN {X 0,Y 475.044,Z 318.658,A -85,B 0,C 180,E1 -7443.178,E2 -7443.178} C_VEL
LIN {X 0,Y 475.236,Z 313.48,A -85,B 0,C 180,E1 -7443.841,E2 -7443.841} C_VEL
LIN {X 0,Y 474.765,Z 309.309,A -85,B 0,C 180,E1 -7444.344,E2 -7444.344} C_VEL
LIN {X 0,Y 472.245,Z 302.344,A -85,B 0,C 180,E1 -7445.148,E2 -7445.148} C_VEL
LIN {X 0,Y 469.784,Z 294.921,A -85,B 0,C 180,E1 -7445.888,E2 -7445.888} C_VEL
LIN {X 0,Y 469.394,Z 290.021,A -85,B 0,C 180,E1 -7446.286,E2 -7446.286} C_VEL
LIN {X 0,Y 469.831,Z 278.248,A -85,B 0,C 180,E1 -7447.055,E2 -7447.055} C_VEL
LIN {X 0,Y 470.262,Z 265.993,A -85,B 0,C 180,E1 -7447.657,E2 -7447.657} C_VEL
LIN {X 0,Y 470.078,Z 262.133,A -85,B 0,C 180,E1 -7447.822,E2 -7447.822} C_VEL
LIN {X 0,Y 467.147,Z 249.613,A -85,B 0,C 180,E1 -7448.314,E2 -7448.314} C_VEL
LIN {X 0,Y 466.819,Z 247.903,A -85,B 0,C 180,E1 -7448.385,E2 -7448.385} C_VEL
LIN {X 0,Y 466.873,Z 244.36,A -85,B 0,C 180,E1 -7451.573,E2 -7451.573} C_VEL
LIN {X 0,Y 466.953,Z 241.244,A -85,B 0,C 180,E1 -7454.41,E2 -7454.41} C_VEL
LIN {X 0,Y 467.032,Z 237.367,A -85,B 0,C 180,E1 -7457.986,E2 -7457.986} C_VEL
LIN {X 0,Y 467.116,Z 233.8,A -85,B 0,C 180,E1 -7461.348,E2 -7461.348} C_VEL
LIN {X 0,Y 467.132,Z 231.009,A -85,B 0,C 180,E1 -7463.956,E2 -7463.956} C_VEL
LIN {X 0,Y 467.221,Z 230.29,A -85,B 0,C 180,E1 -7464.823,E2 -7464.823} C_VEL
LIN {X 0,Y 467.696,Z 230.228,A -85,B 0,C 180,E1 -7468.279,E2 -7468.279} C_VEL
LIN {X 0,Y 467.815,Z 230.215,A -85,B 0,C 180,E1 -7470.862,E2 -7470.862} C_VEL
LIN {X 0,Y 467.847,Z 230.208,A -85,B 0,C 180,E1 -7472.584,E2 -7472.584} C_VEL
LIN {X 0,Y 467.73,Z 230.224,A -85,B 0,C 180,E1 -7476.038,E2 -7476.038} C_VEL
LIN {X 0,Y 467.67,Z 230.231,A -85,B 0,C 180,E1 -7478.644,E2 -7478.644} C_VEL
LIN {X 0,Y 467.684,Z 230.229,A -85,B 0,C 180,E1 -7482.146,E2 -7482.146} C_VEL
LIN {X 0,Y 467.636,Z 230.233,A -85,B 0,C 180,E1 -7485.887,E2 -7485.887} C_VEL
LIN {X 0,Y 467.612,Z 230.239,A -85,B 0,C 180,E1 -7489.309,E2 -7489.309} C_VEL
LIN {X 0,Y 467.538,Z 230.246,A -85,B 0,C 180,E1 -7492.075,E2 -7492.075} C_VEL
LIN {X 0,Y 467.594,Z 230.242,A -85,B 0,C 180,E1 -7494.889,E2 -7494.889} C_VEL
LIN {X 0,Y 467.617,Z 230.237,A -85,B 0,C 180,E1 -7497.77,E2 -7497.77} C_VEL
LIN {X 0,Y 467.559,Z 230.246,A -85,B 0,C 180,E1 -7501.047,E2 -7501.047} C_VEL
LIN {X 0,Y 467.581,Z 230.243,A -85,B 0,C 180,E1 -7504.244,E2 -7504.244} C_VEL
LIN {X 0,Y 467.543,Z 230.248,A -85,B 0,C 180,E1 -7507.189,E2 -7507.189} C_VEL
LIN {X 0,Y 467.589,Z 230.241,A -85,B 0,C 180,E1 -7510.264,E2 -7510.264} C_VEL
LIN {X 0,Y 467.613,Z 230.239,A -85,B 0,C 180,E1 -7512.573,E2 -7512.573} C_VEL
LIN {X 0,Y 467.565,Z 230.245,A -85,B 0,C 180,E1 -7515.055,E2 -7515.055} C_VEL
LIN {X 0,Y 467.584,Z 230.242,A -85,B 0,C 180,E1 -7517.442,E2 -7517.442} C_VEL
LIN {X 0,Y 467.615,Z 230.239,A -85,B 0,C 180,E1 -7520.861,E2 -7520.861} C_VEL
LIN {X 0,Y 467.56,Z 230.246,A -85,B 0,C 180,E1 -7524.262,E2 -7524.262} C_VEL
LIN {X 0,Y 467.58,Z 230.241,A -85,B 0,C 180,E1 -7527.323,E2 -7527.323} C_VEL
LIN {X 0,Y 467.569,Z 230.244,A -85,B 0,C 180,E1 -7530.669,E2 -7530.669} C_VEL
LIN {X 0,Y 467.613,Z 230.237,A -85,B 0,C 180,E1 -7533.201,E2 -7533.201} C_VEL
LIN {X 0,Y 467.592,Z 230.242,A -85,B 0,C 180,E1 -7536.471,E2 -7536.471} C_VEL
LIN {X 0,Y 467.626,Z 230.237,A -85,B 0,C 180,E1 -7539.779,E2 -7539.779} C_VEL
LIN {X 0,Y 467.609,Z 230.24,A -85,B 0,C 180,E1 -7542.508,E2 -7542.508} C_VEL
LIN {X 0,Y 467.61,Z 230.238,A -85,B 0,C 180,E1 -7545.198,E2 -7545.198} C_VEL
LIN {X 0,Y 467.688,Z 230.23,A -85,B 0,C 180,E1 -7547.857,E2 -7547.857} C_VEL
LIN {X 0,Y 467.674,Z 230.23,A -85,B 0,C 180,E1 -7551.359,E2 -7551.359} C_VEL
LIN {X 0,Y 467.747,Z 230.223,A -85,B 0,C 180,E1 -7553.964,E2 -7553.964} C_VEL
LIN {X 0,Y 467.863,Z 230.207,A -85,B 0,C 180,E1 -7557.418,E2 -7557.418} C_VEL
LIN {X 0,Y 467.888,Z 230.205,A -85,B 0,C 180,E1 -7560.001,E2 -7560.001} C_VEL
LIN {X 0,Y 467.858,Z 230.206,A -85,B 0,C 180,E1 -7562.584,E2 -7562.584} C_VEL
LIN {X 0,Y 467.74,Z 230.223,A -85,B 0,C 180,E1 -7566.039,E2 -7566.039} C_VEL
LIN {X 0,Y 467.677,Z 230.229,A -85,B 0,C 180,E1 -7568.644,E2 -7568.644} C_VEL
LIN {X 0,Y 467.665,Z 230.233,A -85,B 0,C 180,E1 -7572.146,E2 -7572.146} C_VEL
LIN {X 0,Y 467.647,Z 230.236,A -85,B 0,C 180,E1 -7575.696,E2 -7575.696} C_VEL
LIN {X 0,Y 467.63,Z 230.238,A -85,B 0,C 180,E1 -7579.309,E2 -7579.309} C_VEL
LIN {X 0,Y 467.543,Z 230.246,A -85,B 0,C 180,E1 -7582.075,E2 -7582.075} C_VEL
LIN {X 0,Y 467.578,Z 230.243,A -85,B 0,C 180,E1 -7584.89,E2 -7584.89} C_VEL
LIN {X 0,Y 467.625,Z 230.236,A -85,B 0,C 180,E1 -7587.77,E2 -7587.77} C_VEL
LIN {X 0,Y 467.577,Z 230.244,A -85,B 0,C 180,E1 -7591.045,E2 -7591.045} C_VEL
LIN {X 0,Y 467.586,Z 230.241,A -85,B 0,C 180,E1 -7594.24,E2 -7594.24} C_VEL
LIN {X 0,Y 467.556,Z 230.246,A -85,B 0,C 180,E1 -7597.186,E2 -7597.186} C_VEL
LIN {X 0,Y 467.583,Z 230.242,A -85,B 0,C 180,E1 -7600.265,E2 -7600.265} C_VEL
LIN {X 0,Y 467.596,Z 230.241,A -85,B 0,C 180,E1 -7602.567,E2 -7602.567} C_VEL
LIN {X 0,Y 467.575,Z 230.241,A -85,B 0,C 180,E1 -7605.053,E2 -7605.053} C_VEL
LIN {X 0,Y 467.598,Z 230.238,A -85,B 0,C 180,E1 -7607.44,E2 -7607.44} C_VEL
LIN {X 0,Y 467.636,Z 230.377,A -85,B 0,C 180,E1 -7609.599,E2 -7609.599} C_VEL
LIN {X 0,Y 468.776,Z 236.979,A -85,B 0,C 180,E1 -7612.618,E2 -7612.618} C_VEL
LIN {X 0,Y 469.17,Z 240.727,A -85,B 0,C 180,E1 -7614.252,E2 -7614.252} C_VEL
LIN {X 0,Y 468.797,Z 248.318,A -85,B 0,C 180,E1 -7617.336,E2 -7617.336} C_VEL
LIN {X 0,Y 468.336,Z 256.44,A -85,B 0,C 180,E1 -7620.502,E2 -7620.502} C_VEL
LIN {X 0,Y 467.879,Z 266.197,A -85,B 0,C 180,E1 -7624.175,E2 -7624.175} C_VEL
LIN {X 0,Y 467.51,Z 275.232,A -85,B 0,C 180,E1 -7627.459,E2 -7627.459} C_VEL
LIN {X 0,Y 467.234,Z 284.301,A -85,B 0,C 180,E1 -7630.675,E2 -7630.675} C_VEL
LIN {X 0,Y 467.078,Z 293.432,A -85,B 0,C 180,E1 -7633.837,E2 -7633.837} C_VEL
LIN {X 0,Y 466.981,Z 295.654,A -85,B 0,C 180,E1 -7634.6,E2 -7634.6} C_VEL
LIN {X 0,Y 468.984,Z 309.737,A -85,B 0,C 180,E1 -7635.041,E2 -7635.041} C_VEL
LIN {X 0,Y 469.857,Z 317.778,A -85,B 0,C 180,E1 -7635.379,E2 -7635.379} C_VEL
LIN {X 0,Y 469.359,Z 330.88,A -85,B 0,C 180,E1 -7636.027,E2 -7636.027} C_VEL
LIN {X 0,Y 468.84,Z 342.339,A -85,B 0,C 180,E1 -7636.784,E2 -7636.784} C_VEL
LIN {X 0,Y 468.315,Z 353.407,A -85,B 0,C 180,E1 -7637.708,E2 -7637.708} C_VEL
LIN {X 0,Y 467.899,Z 363.371,A -85,B 0,C 180,E1 -7638.739,E2 -7638.739} C_VEL
LIN {X 0,Y 467.462,Z 371.943,A -85,B 0,C 180,E1 -7639.824,E2 -7639.824} C_VEL
LIN {X 0,Y 467.117,Z 380.292,A -85,B 0,C 180,E1 -7641.128,E2 -7641.128} C_VEL
LIN {X 0,Y 466.927,Z 387.029,A -85,B 0,C 180,E1 -7642.431,E2 -7642.431} C_VEL
LIN {X 0,Y 466.759,Z 393.199,A -85,B 0,C 180,E1 -7643.949,E2 -7643.949} C_VEL
LIN {X 0,Y 466.693,Z 397.203,A -85,B 0,C 180,E1 -7645.248,E2 -7645.248} C_VEL
LIN {X 0,Y 466.73,Z 400.159,A -85,B 0,C 180,E1 -7646.546,E2 -7646.546} C_VEL
LIN {X 0,Y 466.702,Z 401.565,A -85,B 0,C 180,E1 -7647.41,E2 -7647.41} C_VEL
LIN {X 0,Y 466.694,Z 402.563,A -85,B 0,C 180,E1 -7648.273,E2 -7648.273} C_VEL
LIN {X 0,Y 466.608,Z 403.374,A -85,B 0,C 180,E1 -7649.999,E2 -7649.999} C_VEL
LIN {X 0,Y 466.694,Z 402.526,A -85,B 0,C 180,E1 -7651.725,E2 -7651.725} C_VEL
LIN {X 0,Y 466.702,Z 401.509,A -85,B 0,C 180,E1 -7652.588,E2 -7652.588} C_VEL
LIN {X 0,Y 466.73,Z 400.087,A -85,B 0,C 180,E1 -7653.452,E2 -7653.452} C_VEL
LIN {X 0,Y 466.693,Z 397.097,A -85,B 0,C 180,E1 -7654.75,E2 -7654.75} C_VEL
LIN {X 0,Y 466.753,Z 393.062,A -85,B 0,C 180,E1 -7656.049,E2 -7656.049} C_VEL
LIN {X 0,Y 466.925,Z 386.866,A -85,B 0,C 180,E1 -7657.567,E2 -7657.567} C_VEL
LIN {X 0,Y 467.112,Z 380.102,A -85,B 0,C 180,E1 -7658.871,E2 -7658.871} C_VEL
LIN {X 0,Y 467.437,Z 371.724,A -85,B 0,C 180,E1 -7660.175,E2 -7660.175} C_VEL
LIN {X 0,Y 467.877,Z 363.146,A -85,B 0,C 180,E1 -7661.26,E2 -7661.26} C_VEL
LIN {X 0,Y 468.328,Z 353.288,A -85,B 0,C 180,E1 -7662.28,E2 -7662.28} C_VEL
LIN {X 0,Y 468.792,Z 342.126,A -85,B 0,C 180,E1 -7663.215,E2 -7663.215} C_VEL
LIN {X 0,Y 469.332,Z 330.709,A -85,B 0,C 180,E1 -7663.972,E2 -7663.972} C_VEL
LIN {X 0,Y 469.809,Z 319.012,A -85,B 0,C 180,E1 -7664.566,E2 -7664.566} C_VEL
LIN {X 0,Y 469.209,Z 311.866,A -85,B 0,C 180,E1 -7664.874,E2 -7664.874} C_VEL
LIN {X 0,Y 467.568,Z 298.957,A -85,B 0,C 180,E1 -7665.317,E2 -7665.317} C_VEL
LIN {X 0,Y 466.977,Z 294.945,A -85,B 0,C 180,E1 -7665.445,E2 -7665.445} C_VEL
LIN {X 0,Y 467.175,Z 284.85,A -85,B 0,C 180,E1 -7668.908,E2 -7668.908} C_VEL
LIN {X 0,Y 467.388,Z 277.137,A -85,B 0,C 180,E1 -7671.616,E2 -7671.616} C_VEL
LIN {X 0,Y 467.676,Z 268.083,A -85,B 0,C 180,E1 -7674.882,E2 -7674.882} C_VEL
LIN {X 0,Y 468.045,Z 259.14,A -85,B 0,C 180,E1 -7678.228,E2 -7678.228} C_VEL
LIN {X 0,Y 468.609,Z 250.433,A -85,B 0,C 180,E1 -7681.661,E2 -7681.661} C_VEL
LIN {X 0,Y 469.053,Z 243.078,A -85,B 0,C 180,E1 -7684.705,E2 -7684.705} C_VEL
LIN {X 0,Y 469.133,Z 240.13,A -85,B 0,C 180,E1 -7686.004,E2 -7686.004} C_VEL
